LIN {X 0,Y 358.327,Z 844.562,A -85,B 0,C 180,E1 17293.72,E2 17293.72} C_VEL
LIN {X 0,Y 357.15,Z 856.767,A -85,B 0,C 180,E1 17291.793,E2 17291.793} C_VEL
LIN {X 0,Y 356.13,Z 867.565,A -85,B 0,C 180,E1 17289.698,E2 17289.698} C_VEL
LIN {X 0,Y 355.243,Z 877.441,A -85,B 0,C 180,E1 17287.277,E2 17287.277} C_VEL
LIN {X 0,Y 354.65,Z 885.167,A -85,B 0,C 180,E1 17284.852,E2 17284.852} C_VEL
LIN {X 0,Y 354.297,Z 891.351,A -85,B 0,C 180,E1 17282.265,E2 17282.265} C_VEL
LIN {X 0,Y 354.201,Z 895.635,A -85,B 0,C 180,E1 17279.677,E2 17279.677} C_VEL
LIN {X 0,Y 354.349,Z 898.233,A -85,B 0,C 180,E1 17277.089,E2 17277.089} C_VEL
LIN {X 0,Y 354.713,Z 899.091,A -85,B 0,C 180,E1 17274.501,E2 17274.501} C_VEL
LIN {X 0,Y 355.419,Z 898.216,A -85,B 0,C 180,E1 17271.751,E2 17271.751} C_VEL
LIN {X 0,Y 356.484,Z 895.398,A -85,B 0,C 180,E1 17269.005,E2 17269.005} C_VEL
LIN {X 0,Y 357.89,Z 890.872,A -85,B 0,C 180,E1 17266.428,E2 17266.428} C_VEL
LIN {X 0,Y 359.589,Z 884.914,A -85,B 0,C 180,E1 17264.022,E2 17264.022} C_VEL
LIN {X 0,Y 361.837,Z 876.313,A -85,B 0,C 180,E1 17261.472,E2 17261.472} C_VEL
LIN {X 0,Y 364.2,Z 866.559,A -85,B 0,C 180,E1 17259.259,E2 17259.259} C_VEL
LIN {X 0,Y 366.508,Z 856.117,A -85,B 0,C 180,E1 17257.378,E2 17257.378} C_VEL
LIN {X 0,Y 368.84,Z 844.36,A -85,B 0,C 180,E1 17255.667,E2 17255.667} C_VEL
LIN {X 0,Y 371.242,Z 830.372,A -85,B 0,C 180,E1 17254.046,E2 17254.046} C_VEL
LIN {X 0,Y 373.396,Z 815.063,A -85,B 0,C 180,E1 17252.663,E2 17252.663} C_VEL
LIN {X 0,Y 375.26,Z 798.255,A -85,B 0,C 180,E1 17251.515,E2 17251.515} C_VEL
LIN {X 0,Y 379.041,Z 772.114,A -85,B 0,C 180,E1 17250.009,E2 17250.009} C_VEL
LIN {X 0,Y 387.538,Z 729.748,A -85,B 0,C 180,E1 17247.894,E2 17247.894} C_VEL
LIN {X 0,Y 397.033,Z 682.025,A -85,B 0,C 180,E1 17245.846,E2 17245.846} C_VEL
LIN {X 0,Y 397.784,Z 679.73,A -85,B 0,C 180,E1 17245.734,E2 17245.734} C_VEL
LIN {X 0,Y 407.089,Z 665.776,A -85,B 0,C 180,E1 17244.661,E2 17244.661} C_VEL
LIN {X 0,Y 408.416,Z 663.697,A -85,B 0,C 180,E1 17244.363,E2 17244.363} C_VEL
LIN {X 0,Y 415.736,Z 652.988,A -85,B 0,C 180,E1 17242.392,E2 17242.392} C_VEL
LIN {X 0,Y 409.908,Z 662.726,A -85,B 0,C 180,E1 17240.427,E2 17240.427} C_VEL
LIN {X 0,Y 406.103,Z 673.236,A -85,B 0,C 180,E1 17238.247,E2 17238.247} C_VEL
LIN {X 0,Y 404.763,Z 684.168,A -85,B 0,C 180,E1 17235.96,E2 17235.96} C_VEL
LIN {X 0,Y 406.043,Z 694.968,A -85,B 0,C 180,E1 17233.72,E2 17233.72} C_VEL
LIN {X 0,Y 408.323,Z 702.84,A -85,B 0,C 180,E1 17232.141,E2 17232.141} C_VEL
LIN {X 0,Y 398.65,Z 721.921,A -85,B 0,C 180,E1 17231.177,E2 17231.177} C_VEL
LIN {X 0,Y 396.234,Z 727.339,A -85,B 0,C 180,E1 17230.919,E2 17230.919} C_VEL
LIN {X 0,Y 391.082,Z 751.783,A -85,B 0,C 180,E1 17230.609,E2 17230.609} C_VEL
LIN {X 0,Y 389.402,Z 762.099,A -85,B 0,C 180,E1 17230.457,E2 17230.457} C_VEL
LIN {X 0,Y 387.915,Z 782.543,A -85,B 0,C 180,E1 17230.159,E2 17230.159} C_VEL
LIN {X 0,Y 386.621,Z 805.179,A -85,B 0,C 180,E1 17229.634,E2 17229.634} C_VEL
LIN {X 0,Y 384.476,Z 826.222,A -85,B 0,C 180,E1 17228.907,E2 17228.907} C_VEL
LIN {X 0,Y 381.713,Z 846.978,A -85,B 0,C 180,E1 17227.898,E2 17227.898} C_VEL
LIN {X 0,Y 378.758,Z 865.544,A -85,B 0,C 180,E1 17226.722,E2 17226.722} C_VEL
LIN {X 0,Y 375.32,Z 884.39,A -85,B 0,C 180,E1 17225.224,E2 17225.224} C_VEL
LIN {X 0,Y 371.531,Z 902.981,A -85,B 0,C 180,E1 17223.392,E2 17223.392} C_VEL
LIN {X 0,Y 367.741,Z 920.372,A -85,B 0,C 180,E1 17221.287,E2 17221.287} C_VEL
LIN {X 0,Y 364.185,Z 936.094,A -85,B 0,C 180,E1 17218.986,E2 17218.986} C_VEL
LIN {X 0,Y 360.968,Z 950.344,A -85,B 0,C 180,E1 17216.486,E2 17216.486} C_VEL
LIN {X 0,Y 358.088,Z 963.562,A -85,B 0,C 180,E1 17213.709,E2 17213.709} C_VEL
LIN {X 0,Y 355.694,Z 975.773,A -85,B 0,C 180,E1 17210.6,E2 17210.6} C_VEL
LIN {X 0,Y 353.976,Z 985.945,A -85,B 0,C 180,E1 17207.423,E2 17207.423} C_VEL
LIN {X 0,Y 352.891,Z 994.085,A -85,B 0,C 180,E1 17204.271,E2 17204.271} C_VEL
LIN {X 0,Y 352.346,Z 1000.464,A -85,B 0,C 180,E1 17201.127,E2 17201.127} C_VEL
LIN {X 0,Y 352.156,Z 1005.337,A -85,B 0,C 180,E1 17197.834,E2 17197.834} C_VEL
LIN {X 0,Y 352.163,Z 1008.374,A -85,B 0,C 180,E1 17194.724,E2 17194.724} C_VEL
LIN {X 0,Y 352.223,Z 1009.946,A -85,B 0,C 180,E1 17191.628,E2 17191.628} C_VEL
LIN {X 0,Y 352.225,Z 1009.994,A -85,B 0,C 180,E1 17188.7,E2 17188.7} C_VEL
LIN {X 0,Y 352.165,Z 1008.606,A -85,B 0,C 180,E1 17185.604,E2 17185.604} C_VEL
LIN {X 0,Y 352.117,Z 1005.756,A -85,B 0,C 180,E1 17182.495,E2 17182.495} C_VEL
LIN {X 0,Y 352.294,Z 1001.017,A -85,B 0,C 180,E1 17179.205,E2 17179.205} C_VEL
LIN {X 0,Y 352.795,Z 994.807,A -85,B 0,C 180,E1 17176.061,E2 17176.061} C_VEL
LIN {X 0,Y 353.805,Z 986.872,A -85,B 0,C 180,E1 17172.909,E2 17172.909} C_VEL
LIN {X 0,Y 355.418,Z 977.017,A -85,B 0,C 180,E1 17169.757,E2 17169.757} C_VEL
LIN {X 0,Y 357.478,Z 966.389,A -85,B 0,C 180,E1 17166.948,E2 17166.948} C_VEL
LIN {X 0,Y 360.351,Z 953.009,A -85,B 0,C 180,E1 17164.026,E2 17164.026} C_VEL
LIN {X 0,Y 363.681,Z 938.075,A -85,B 0,C 180,E1 17161.332,E2 17161.332} C_VEL
LIN {X 0,Y 367.303,Z 922.064,A -85,B 0,C 180,E1 17158.947,E2 17158.947} C_VEL
LIN {X 0,Y 370.863,Z 905.617,A -85,B 0,C 180,E1 17156.912,E2 17156.912} C_VEL
LIN {X 0,Y 374.426,Z 888.379,A -85,B 0,C 180,E1 17155.149,E2 17155.149} C_VEL
LIN {X 0,Y 377.967,Z 869.449,A -85,B 0,C 180,E1 17153.568,E2 17153.568} C_VEL
LIN {X 0,Y 381.074,Z 850.673,A -85,B 0,C 180,E1 17152.314,E2 17152.314} C_VEL
LIN {X 0,Y 383.853,Z 830.914,A -85,B 0,C 180,E1 17151.292,E2 17151.292} C_VEL
LIN {X 0,Y 386.143,Z 809.808,A -85,B 0,C 180,E1 17150.496,E2 17150.496} C_VEL
LIN {X 0,Y 387.604,Z 787.894,A -85,B 0,C 180,E1 17149.946,E2 17149.946} C_VEL
LIN {X 0,Y 388.886,Z 765.567,A -85,B 0,C 180,E1 17149.574,E2 17149.574} C_VEL
LIN {X 0,Y 392.068,Z 738.697,A -85,B 0,C 180,E1 17149.337,E2 17149.337} C_VEL
LIN {X 0,Y 394.002,Z 728.374,A -85,B 0,C 180,E1 17149.294,E2 17149.294} C_VEL
LIN {X 0,Y 406.256,Z 703.937,A -85,B 0,C 180,E1 17147.978,E2 17147.978} C_VEL
LIN {X 0,Y 407.296,Z 701.642,A -85,B 0,C 180,E1 17147.848,E2 17147.848} C_VEL
LIN {X 0,Y 400.592,Z 686.213,A -85,B 0,C 180,E1 17145.753,E2 17145.753} C_VEL
LIN {X 0,Y 395.618,Z 668.635,A -85,B 0,C 180,E1 17143.504,E2 17143.504} C_VEL
LIN {X 0,Y 392.777,Z 649.847,A -85,B 0,C 180,E1 17141.247,E2 17141.247} C_VEL
LIN {X 0,Y 392.112,Z 630.144,A -85,B 0,C 180,E1 17139.038,E2 17139.038} C_VEL
LIN {X 0,Y 393.724,Z 606.831,A -85,B 0,C 180,E1 17136.634,E2 17136.634} C_VEL
LIN {X 0,Y 400.166,Z 566.042,A -85,B 0,C 180,E1 17132.748,E2 17132.748} C_VEL
LIN {X 0,Y 391.222,Z 546.366,A -85,B 0,C 180,E1 17129.051,E2 17129.051} C_VEL
LIN {X 0,Y 382.764,Z 528.585,A -85,B 0,C 180,E1 17125.366,E2 17125.366} C_VEL
LIN {X 0,Y 374.331,Z 511.509,A -85,B 0,C 180,E1 17121.465,E2 17121.465} C_VEL
LIN {X 0,Y 367.669,Z 498.547,A -85,B 0,C 180,E1 17118.224,E2 17118.224} C_VEL
LIN {X 0,Y 362.734,Z 489.046,A -85,B 0,C 180,E1 17115.672,E2 17115.672} C_VEL
LIN {X 0,Y 360.463,Z 484.681,A -85,B 0,C 180,E1 17114.456,E2 17114.456} C_VEL
LIN {X 0,Y 357.931,Z 479.938,A -85,B 0,C 180,E1 17113.077,E2 17113.077} C_VEL
LIN {X 0,Y 355.754,Z 475.696,A -85,B 0,C 180,E1 17111.839,E2 17111.839} C_VEL
LIN {X 0,Y 354.097,Z 472.685,A -85,B 0,C 180,E1 17110.905,E2 17110.905} C_VEL
LIN {X 0,Y 353.827,Z 471.413,A -85,B 0,C 180,E1 17110.584,E2 17110.584} C_VEL
LIN {X 0,Y 353.868,Z 471.408,A -85,B 0,C 180,E1 17106.489,E2 17106.489} C_VEL
LIN {X 0,Y 353.825,Z 471.412,A -85,B 0,C 180,E1 17102.267,E2 17102.267} C_VEL
LIN {X 0,Y 353.866,Z 471.403,A -85,B 0,C 180,E1 17098.219,E2 17098.219} C_VEL
LIN {X 0,Y 353.825,Z 471.407,A -85,B 0,C 180,E1 17093.998,E2 17093.998} C_VEL
LIN {X 0,Y 353.864,Z 471.405,A -85,B 0,C 180,E1 17089.91,E2 17089.91} C_VEL
LIN {X 0,Y 353.822,Z 471.397,A -85,B 0,C 180,E1 17085.6,E2 17085.6} C_VEL
LIN {X 0,Y 353.864,Z 471.384,A -85,B 0,C 180,E1 17081.551,E2 17081.551} C_VEL
LIN {X 0,Y 353.822,Z 471.39,A -85,B 0,C 180,E1 17077.398,E2 17077.398} C_VEL
LIN {X 0,Y 353.865,Z 471.389,A -85,B 0,C 180,E1 17073.234,E2 17073.234} C_VEL
LIN {X 0,Y 353.823,Z 471.397,A -85,B 0,C 180,E1 17069.048,E2 17069.048} C_VEL
LIN {X 0,Y 353.862,Z 471.507,A -85,B 0,C 180,E1 17067.193,E2 17067.193} C_VEL
LIN {X 0,Y 355.032,Z 474.666,A -85,B 0,C 180,E1 17066.47,E2 17066.47} C_VEL
LIN {X 0,Y 356.9,Z 476.875,A -85,B 0,C 180,E1 17065.729,E2 17065.729} C_VEL
LIN {X 0,Y 358.818,Z 480.752,A -85,B 0,C 180,E1 17064.773,E2 17064.773} C_VEL
LIN {X 0,Y 359.911,Z 482.426,A -85,B 0,C 180,E1 17064.31,E2 17064.31} C_VEL
LIN {X 0,Y 365.518,Z 492.86,A -85,B 0,C 180,E1 17061.814,E2 17061.814} C_VEL
LIN {X 0,Y 371.605,Z 504.363,A -85,B 0,C 180,E1 17059.328,E2 17059.328} C_VEL
LIN {X 0,Y 382.76,Z 521.472,A -85,B 0,C 180,E1 17056.939,E2 17056.939} C_VEL
LIN {X 0,Y 393.149,Z 539.114,A -85,B 0,C 180,E1 17054.878,E2 17054.878} C_VEL
LIN {X 0,Y 397.29,Z 547.107,A -85,B 0,C 180,E1 17054.083,E2 17054.083} C_VEL
LIN {X 0,Y 388.766,Z 764.74,A -85,B 0,C 180,E1 17049.883,E2 17049.883} C_VEL
LIN {X 0,Y 387.23,Z 785.322,A -85,B 0,C 180,E1 17049.247,E2 17049.247} C_VEL
LIN {X 0,Y 385.016,Z 805.804,A -85,B 0,C 180,E1 17048.346,E2 17048.346} C_VEL
LIN {X 0,Y 382.432,Z 824.71,A -85,B 0,C 180,E1 17047.246,E2 17047.246} C_VEL
LIN {X 0,Y 379.409,Z 843.123,A -85,B 0,C 180,E1 17045.898,E2 17045.898} C_VEL
LIN {X 0,Y 375.891,Z 861.453,A -85,B 0,C 180,E1 17044.234,E2 17044.234} C_VEL
LIN {X 0,Y 372.225,Z 878.68,A -85,B 0,C 180,E1 17042.312,E2 17042.312} C_VEL
LIN {X 0,Y 368.616,Z 894.311,A -85,B 0,C 180,E1 17040.208,E2 17040.208} C_VEL
LIN {X 0,Y 365.189,Z 908.557,A -85,B 0,C 180,E1 17037.916,E2 17037.916} C_VEL
LIN {X 0,Y 361.934,Z 921.884,A -85,B 0,C 180,E1 17035.352,E2 17035.352} C_VEL
LIN {X 0,Y 359.073,Z 933.808,A -85,B 0,C 180,E1 17032.597,E2 17032.597} C_VEL
LIN {X 0,Y 356.646,Z 944.461,A -85,B 0,C 180,E1 17029.613,E2 17029.613} C_VEL
LIN {X 0,Y 354.714,Z 953.775,A -85,B 0,C 180,E1 17026.371,E2 17026.371} C_VEL
LIN {X 0,Y 353.405,Z 961.197,A -85,B 0,C 180,E1 17023.081,E2 17023.081} C_VEL
LIN {X 0,Y 352.629,Z 966.798,A -85,B 0,C 180,E1 17019.794,E2 17019.794} C_VEL
LIN {X 0,Y 352.248,Z 970.723,A -85,B 0,C 180,E1 17016.519,E2 17016.519} C_VEL
LIN {X 0,Y 352.161,Z 971.831,A -85,B 0,C 180,E1 17015.277,E2 17015.277} C_VEL
LIN {X 0,Y 351.121,Z 972.736,A -85,B 0,C 180,E1 17014.032,E2 17014.032} C_VEL
LIN {X 0,Y 346.458,Z 973.982,A -85,B 0,C 180,E1 17011.675,E2 17011.675} C_VEL
LIN {X 0,Y 344.214,Z 974.308,A -85,B 0,C 180,E1 17010.044,E2 17010.044} C_VEL
LIN {X 0,Y 344.066,Z 974.269,A -85,B 0,C 180,E1 17009.579,E2 17009.579} C_VEL
LIN {X 0,Y 344.109,Z 973.398,A -85,B 0,C 180,E1 17006.334,E2 17006.334} C_VEL
LIN {X 0,Y 344.298,Z 970.92,A -85,B 0,C 180,E1 17002.993,E2 17002.993} C_VEL
LIN {X 0,Y 344.737,Z 966.862,A -85,B 0,C 180,E1 16999.64,E2 16999.64} C_VEL
LIN {X 0,Y 345.615,Z 961.121,A -85,B 0,C 180,E1 16996.276,E2 16996.276} C_VEL
LIN {X 0,Y 346.993,Z 953.972,A -85,B 0,C 180,E1 16993.07,E2 16993.07} C_VEL
LIN {X 0,Y 348.982,Z 945.03,A -85,B 0,C 180,E1 16989.89,E2 16989.89} C_VEL
LIN {X 0,Y 351.675,Z 933.95,A -85,B 0,C 180,E1 16986.721,E2 16986.721} C_VEL
LIN {X 0,Y 354.725,Z 921.962,A -85,B 0,C 180,E1 16983.913,E2 16983.913} C_VEL
LIN {X 0,Y 358.171,Z 908.563,A -85,B 0,C 180,E1 16981.304,E2 16981.304} C_VEL
LIN {X 0,Y 361.933,Z 893.686,A -85,B 0,C 180,E1 16978.895,E2 16978.895} C_VEL
LIN {X 0,Y 365.672,Z 878.113,A -85,B 0,C 180,E1 16976.793,E2 16976.793} C_VEL
LIN {X 0,Y 369.445,Z 861.121,A -85,B 0,C 180,E1 16974.892,E2 16974.892} C_VEL
LIN {X 0,Y 373.11,Z 842.762,A -85,B 0,C 180,E1 16973.215,E2 16973.215} C_VEL
LIN {X 0,Y 376.295,Z 824.075,A -85,B 0,C 180,E1 16971.845,E2 16971.845} C_VEL
LIN {X 0,Y 379.033,Z 804.56,A -85,B 0,C 180,E1 16970.72,E2 16970.72} C_VEL
LIN {X 0,Y 381.218,Z 784.635,A -85,B 0,C 180,E1 16969.854,E2 16969.854} C_VEL
LIN {X 0,Y 382.807,Z 763.298,A -85,B 0,C 180,E1 16969.208,E2 16969.208} C_VEL
LIN {X 0,Y 391.184,Z 555.703,A -85,B 0,C 180,E1 16965.148,E2 16965.148} C_VEL
LIN {X 0,Y 382.835,Z 539.982,A -85,B 0,C 180,E1 16963.461,E2 16963.461} C_VEL
LIN {X 0,Y 372.499,Z 522.649,A -85,B 0,C 180,E1 16961.247,E2 16961.247} C_VEL
LIN {X 0,Y 368.988,Z 517.5,A -85,B 0,C 180,E1 16960.465,E2 16960.465} C_VEL
LIN {X 0,Y 366.654,Z 518.374,A -85,B 0,C 180,E1 16960.059,E2 16960.059} C_VEL
LIN {X 0,Y 364.475,Z 517.811,A -85,B 0,C 180,E1 16959.629,E2 16959.629} C_VEL
LIN {X 0,Y 364.222,Z 517.629,A -85,B 0,C 180,E1 16959.56,E2 16959.56} C_VEL
LIN {X 0,Y 370.358,Z 535.71,A -85,B 0,C 180,E1 16956.174,E2 16956.174} C_VEL
LIN {X 0,Y 371.873,Z 541.268,A -85,B 0,C 180,E1 16955.221,E2 16955.221} C_VEL
LIN {X 0,Y 367.71,Z 575.018,A -85,B 0,C 180,E1 16951.107,E2 16951.107} C_VEL
LIN {X 0,Y 363.77,Z 611.009,A -85,B 0,C 180,E1 16946.793,E2 16946.793} C_VEL
LIN {X 0,Y 361.959,Z 630.785,A -85,B 0,C 180,E1 16944.502,E2 16944.502} C_VEL
LIN {X 0,Y 362.358,Z 637.138,A -85,B 0,C 180,E1 16944.255,E2 16944.255} C_VEL
LIN {X 0,Y 355.628,Z 765.283,A -85,B 0,C 180,E1 16940.307,E2 16940.307} C_VEL
LIN {X 0,Y 355.062,Z 783.346,A -85,B 0,C 180,E1 16939.585,E2 16939.585} C_VEL
LIN {X 0,Y 354.204,Z 800.194,A -85,B 0,C 180,E1 16938.602,E2 16938.602} C_VEL
LIN {X 0,Y 353.149,Z 815.686,A -85,B 0,C 180,E1 16937.38,E2 16937.38} C_VEL
LIN {X 0,Y 351.952,Z 830.328,A -85,B 0,C 180,E1 16935.911,E2 16935.911} C_VEL
LIN {X 0,Y 350.574,Z 845.108,A -85,B 0,C 180,E1 16934.03,E2 16934.03} C_VEL
LIN {X 0,Y 349.35,Z 857.47,A -85,B 0,C 180,E1 16932.06,E2 16932.06} C_VEL
LIN {X 0,Y 348.283,Z 868.348,A -85,B 0,C 180,E1 16929.919,E2 16929.919} C_VEL
LIN {X 0,Y 347.408,Z 877.732,A -85,B 0,C 180,E1 16927.608,E2 16927.608} C_VEL
LIN {X 0,Y 346.779,Z 885.724,A -85,B 0,C 180,E1 16925.128,E2 16925.128} C_VEL
LIN {X 0,Y 346.389,Z 892.109,A -85,B 0,C 180,E1 16922.482,E2 16922.482} C_VEL
LIN {X 0,Y 346.293,Z 896.653,A -85,B 0,C 180,E1 16919.835,E2 16919.835} C_VEL
LIN {X 0,Y 346.458,Z 899.551,A -85,B 0,C 180,E1 16917.023,E2 16917.023} C_VEL
LIN {X 0,Y 346.867,Z 900.541,A -85,B 0,C 180,E1 16914.376,E2 16914.376} C_VEL
LIN {X 0,Y 347.635,Z 899.778,A -85,B 0,C 180,E1 16911.565,E2 16911.565} C_VEL
LIN {X 0,Y 348.881,Z 896.874,A -85,B 0,C 180,E1 16908.595,E2 16908.595} C_VEL
LIN {X 0,Y 350.434,Z 892.375,A -85,B 0,C 180,E1 16905.955,E2 16905.955} C_VEL
LIN {X 0,Y 352.411,Z 885.971,A -85,B 0,C 180,E1 16903.348,E2 16903.348} C_VEL
LIN {X 0,Y 354.739,Z 877.962,A -85,B 0,C 180,E1 16900.916,E2 16900.916} C_VEL
LIN {X 0,Y 357.498,Z 867.558,A -85,B 0,C 180,E1 16898.508,E2 16898.508} C_VEL
LIN {X 0,Y 360.338,Z 855.603,A -85,B 0,C 180,E1 16896.362,E2 16896.362} C_VEL
LIN {X 0,Y 363.15,Z 842.283,A -85,B 0,C 180,E1 16894.476,E2 16894.476} C_VEL
LIN {X 0,Y 365.813,Z 827.572,A -85,B 0,C 180,E1 16892.842,E2 16892.842} C_VEL
LIN {X 0,Y 368.218,Z 811.346,A -85,B 0,C 180,E1 16891.451,E2 16891.451} C_VEL
LIN {X 0,Y 371.798,Z 786.102,A -85,B 0,C 180,E1 16889.809,E2 16889.809} C_VEL
LIN {X 0,Y 378.125,Z 755.401,A -85,B 0,C 180,E1 16888.072,E2 16888.072} C_VEL
LIN {X 0,Y 388.531,Z 709.223,A -85,B 0,C 180,E1 16885.875,E2 16885.875} C_VEL
LIN {X 0,Y 394.034,Z 683.55,A -85,B 0,C 180,E1 16884.794,E2 16884.794} C_VEL
LIN {X 0,Y 403.144,Z 670.374,A -85,B 0,C 180,E1 16883.824,E2 16883.824} C_VEL
LIN {X 0,Y 404.573,Z 668.344,A -85,B 0,C 180,E1 16883.621,E2 16883.621} C_VEL
LIN {X 0,Y 409.42,Z 661.58,A -85,B 0,C 180,E1 16882.355,E2 16882.355} C_VEL
LIN {X 0,Y 403.832,Z 671.327,A -85,B 0,C 180,E1 16880.299,E2 16880.299} C_VEL
LIN {X 0,Y 400.331,Z 682.047,A -85,B 0,C 180,E1 16877.983,E2 16877.983} C_VEL
LIN {X 0,Y 399.464,Z 692.505,A -85,B 0,C 180,E1 16875.707,E2 16875.707} C_VEL
LIN {X 0,Y 401.087,Z 702.877,A -85,B 0,C 180,E1 16873.476,E2 16873.476} C_VEL
LIN {X 0,Y 401.753,Z 705.735,A -85,B 0,C 180,E1 16872.897,E2 16872.897} C_VEL
LIN {X 0,Y 392.641,Z 724.079,A -85,B 0,C 180,E1 16871.958,E2 16871.958} C_VEL
LIN {X 0,Y 386.129,Z 754.105,A -85,B 0,C 180,E1 16871.548,E2 16871.548} C_VEL
LIN {X 0,Y 382.336,Z 772.967,A -85,B 0,C 180,E1 16871.095,E2 16871.095} C_VEL
LIN {X 0,Y 380.859,Z 800.177,A -85,B 0,C 180,E1 16870.537,E2 16870.537} C_VEL
LIN {X 0,Y 378.856,Z 821.051,A -85,B 0,C 180,E1 16869.871,E2 16869.871} C_VEL
LIN {X 0,Y 376.169,Z 841.391,A -85,B 0,C 180,E1 16868.949,E2 16868.949} C_VEL
LIN {X 0,Y 373.036,Z 860.888,A -85,B 0,C 180,E1 16867.768,E2 16867.768} C_VEL
LIN {X 0,Y 369.564,Z 879.545,A -85,B 0,C 180,E1 16866.336,E2 16866.336} C_VEL
LIN {X 0,Y 365.687,Z 898.153,A -85,B 0,C 180,E1 16864.566,E2 16864.566} C_VEL
LIN {X 0,Y 361.789,Z 915.443,A -85,B 0,C 180,E1 16862.551,E2 16862.551} C_VEL
LIN {X 0,Y 358.126,Z 931.067,A -85,B 0,C 180,E1 16860.355,E2 16860.355} C_VEL
LIN {X 0,Y 354.644,Z 945.642,A -85,B 0,C 180,E1 16857.906,E2 16857.906} C_VEL
LIN {X 0,Y 351.397,Z 959.56,A -85,B 0,C 180,E1 16855.086,E2 16855.086} C_VEL
LIN {X 0,Y 348.707,Z 971.862,A -85,B 0,C 180,E1 16852.064,E2 16852.064} C_VEL
LIN {X 0,Y 346.719,Z 982.059,A -85,B 0,C 180,E1 16849.019,E2 16849.019} C_VEL
LIN {X 0,Y 345.336,Z 990.862,A -85,B 0,C 180,E1 16845.794,E2 16845.794} C_VEL
LIN {X 0,Y 344.516,Z 998.173,A -85,B 0,C 180,E1 16842.403,E2 16842.403} C_VEL
LIN {X 0,Y 344.187,Z 1003.425,A -85,B 0,C 180,E1 16839.195,E2 16839.195} C_VEL
LIN {X 0,Y 344.149,Z 1007.041,A -85,B 0,C 180,E1 16836.004,E2 16836.004} C_VEL
LIN {X 0,Y 344.208,Z 1009.106,A -85,B 0,C 180,E1 16832.831,E2 16832.831} C_VEL
LIN {X 0,Y 344.244,Z 1009.723,A -85,B 0,C 180,E1 16829.668,E2 16829.668} C_VEL
LIN {X 0,Y 344.196,Z 1008.891,A -85,B 0,C 180,E1 16826.67,E2 16826.67} C_VEL
LIN {X 0,Y 344.145,Z 1006.54,A -85,B 0,C 180,E1 16823.495,E2 16823.495} C_VEL
LIN {X 0,Y 344.219,Z 1002.436,A -85,B 0,C 180,E1 16820.133,E2 16820.133} C_VEL
LIN {X 0,Y 344.605,Z 996.915,A -85,B 0,C 180,E1 16816.921,E2 16816.921} C_VEL
LIN {X 0,Y 345.55,Z 989.188,A -85,B 0,C 180,E1 16813.528,E2 16813.528} C_VEL
LIN {X 0,Y 347.065,Z 979.934,A -85,B 0,C 180,E1 16810.303,E2 16810.303} C_VEL
LIN {X 0,Y 349.235,Z 969.022,A -85,B 0,C 180,E1 16807.202,E2 16807.202} C_VEL
LIN {X 0,Y 352.042,Z 956.398,A -85,B 0,C 180,E1 16804.245,E2 16804.245} C_VEL
LIN {X 0,Y 355.234,Z 942.818,A -85,B 0,C 180,E1 16801.598,E2 16801.598} C_VEL
LIN {X 0,Y 358.829,Z 927.815,A -85,B 0,C 180,E1 16799.157,E2 16799.157} C_VEL
LIN {X 0,Y 362.69,Z 911.261,A -85,B 0,C 180,E1 16796.919,E2 16796.919} C_VEL
LIN {X 0,Y 366.607,Z 893.632,A -85,B 0,C 180,E1 16794.964,E2 16794.964} C_VEL
LIN {X 0,Y 370.389,Z 874.916,A -85,B 0,C 180,E1 16793.279,E2 16793.279} C_VEL
LIN {X 0,Y 373.723,Z 856.216,A -85,B 0,C 180,E1 16791.927,E2 16791.927} C_VEL
LIN {X 0,Y 376.714,Z 836.78,A -85,B 0,C 180,E1 16790.826,E2 16790.826} C_VEL
LIN {X 0,Y 379.295,Z 816.001,A -85,B 0,C 180,E1 16789.951,E2 16789.951} C_VEL
LIN {X 0,Y 381.074,Z 795.371,A -85,B 0,C 180,E1 16789.345,E2 16789.345} C_VEL
LIN {X 0,Y 382.505,Z 769.105,A -85,B 0,C 180,E1 16788.848,E2 16788.848} C_VEL
LIN {X 0,Y 385.797,Z 739.934,A -85,B 0,C 180,E1 16788.569,E2 16788.569} C_VEL
LIN {X 0,Y 388.428,Z 725.254,A -85,B 0,C 180,E1 16788.534,E2 16788.534} C_VEL
LIN {X 0,Y 399.359,Z 703.372,A -85,B 0,C 180,E1 16787.325,E2 16787.325} C_VEL
LIN {X 0,Y 392.97,Z 687.667,A -85,B 0,C 180,E1 16785.189,E2 16785.189} C_VEL
LIN {X 0,Y 388.217,Z 669.39,A -85,B 0,C 180,E1 16782.838,E2 16782.838} C_VEL
LIN {X 0,Y 385.707,Z 649.996,A -85,B 0,C 180,E1 16780.493,E2 16780.493} C_VEL
LIN {X 0,Y 385.416,Z 629.38,A -85,B 0,C 180,E1 16778.183,E2 16778.183} C_VEL
LIN {X 0,Y 387.601,Z 604.874,A -85,B 0,C 180,E1 16775.653,E2 16775.653} C_VEL
LIN {X 0,Y 393.478,Z 569.598,A -85,B 0,C 180,E1 16772.251,E2 16772.251} C_VEL
LIN {X 0,Y 384.721,Z 550.197,A -85,B 0,C 180,E1 16768.548,E2 16768.548} C_VEL
LIN {X 0,Y 376.279,Z 532.557,A -85,B 0,C 180,E1 16764.824,E2 16764.824} C_VEL
LIN {X 0,Y 368.499,Z 516.647,A -85,B 0,C 180,E1 16761.154,E2 16761.154} C_VEL
LIN {X 0,Y 361.87,Z 503.689,A -85,B 0,C 180,E1 16757.86,E2 16757.86} C_VEL
LIN {X 0,Y 356.908,Z 494.103,A -85,B 0,C 180,E1 16755.268,E2 16755.268} C_VEL
LIN {X 0,Y 352.715,Z 485.947,A -85,B 0,C 180,E1 16752.941,E2 16752.941} C_VEL
LIN {X 0,Y 350.217,Z 481.279,A -85,B 0,C 180,E1 16751.528,E2 16751.528} C_VEL
LIN {X 0,Y 347.771,Z 476.632,A -85,B 0,C 180,E1 16750.1,E2 16750.1} C_VEL
LIN {X 0,Y 346.169,Z 473.606,A -85,B 0,C 180,E1 16749.14,E2 16749.14} C_VEL
LIN {X 0,Y 345.916,Z 472.397,A -85,B 0,C 180,E1 16748.812,E2 16748.812} C_VEL
LIN {X 0,Y 345.91,Z 472.397,A -85,B 0,C 180,E1 16744.642,E2 16744.642} C_VEL
LIN {X 0,Y 345.917,Z 472.394,A -85,B 0,C 180,E1 16740.165,E2 16740.165} C_VEL
LIN {X 0,Y 345.892,Z 472.395,A -85,B 0,C 180,E1 16736.022,E2 16736.022} C_VEL
LIN {X 0,Y 345.917,Z 472.369,A -85,B 0,C 180,E1 16731.69,E2 16731.69} C_VEL
LIN {X 0,Y 345.891,Z 472.377,A -85,B 0,C 180,E1 16727.648,E2 16727.648} C_VEL
LIN {X 0,Y 345.919,Z 472.385,A -85,B 0,C 180,E1 16723.372,E2 16723.372} C_VEL
LIN {X 0,Y 345.891,Z 472.4,A -85,B 0,C 180,E1 16719.172,E2 16719.172} C_VEL
LIN {X 0,Y 345.926,Z 472.397,A -85,B 0,C 180,E1 16714.856,E2 16714.856} C_VEL
LIN {X 0,Y 345.897,Z 472.4,A -85,B 0,C 180,E1 16710.567,E2 16710.567} C_VEL
LIN {X 0,Y 345.888,Z 472.397,A -85,B 0,C 180,E1 16709.151,E2 16709.151} C_VEL
LIN {X 0,Y 347.044,Z 475.6,A -85,B 0,C 180,E1 16708.375,E2 16708.375} C_VEL
LIN {X 0,Y 349.2,Z 478.304,A -85,B 0,C 180,E1 16707.432,E2 16707.432} C_VEL
LIN {X 0,Y 351.081,Z 481.889,A -85,B 0,C 180,E1 16706.461,E2 16706.461} C_VEL
LIN {X 0,Y 352.18,Z 483.366,A -85,B 0,C 180,E1 16705.993,E2 16705.993} C_VEL
LIN {X 0,Y 357.956,Z 493.917,A -85,B 0,C 180,E1 16703.288,E2 16703.288} C_VEL
LIN {X 0,Y 364.46,Z 505.727,A -85,B 0,C 180,E1 16700.623,E2 16700.623} C_VEL
LIN {X 0,Y 375.385,Z 522.241,A -85,B 0,C 180,E1 16698.147,E2 16698.147} C_VEL
LIN {X 0,Y 386.228,Z 540.302,A -85,B 0,C 180,E1 16695.888,E2 16695.888} C_VEL
LIN {X 0,Y 391.461,Z 550.328,A -85,B 0,C 180,E1 16694.84,E2 16694.84} C_VEL
LIN {X 0,Y 382.655,Z 765.265,A -85,B 0,C 180,E1 16690.646,E2 16690.646} C_VEL
LIN {X 0,Y 381.071,Z 785.681,A -85,B 0,C 180,E1 16690.008,E2 16690.008} C_VEL
LIN {X 0,Y 378.76,Z 806.255,A -85,B 0,C 180,E1 16689.094,E2 16689.094} C_VEL
LIN {X 0,Y 376.08,Z 825.101,A -85,B 0,C 180,E1 16687.985,E2 16687.985} C_VEL
LIN {X 0,Y 372.929,Z 843.521,A -85,B 0,C 180,E1 16686.622,E2 16686.622} C_VEL
LIN {X 0,Y 369.262,Z 861.856,A -85,B 0,C 180,E1 16684.937,E2 16684.937} C_VEL
LIN {X 0,Y 365.426,Z 879.088,A -85,B 0,C 180,E1 16682.989,E2 16682.989} C_VEL
LIN {X 0,Y 361.663,Z 894.667,A -85,B 0,C 180,E1 16680.861,E2 16680.861} C_VEL
LIN {X 0,Y 358.042,Z 908.971,A -85,B 0,C 180,E1 16678.523,E2 16678.523} C_VEL
LIN {X 0,Y 354.616,Z 922.3,A -85,B 0,C 180,E1 16675.914,E2 16675.914} C_VEL
LIN {X 0,Y 351.588,Z 934.225,A -85,B 0,C 180,E1 16673.106,E2 16673.106} C_VEL
LIN {X 0,Y 348.943,Z 945.143,A -85,B 0,C 180,E1 16669.973,E2 16669.973} C_VEL
LIN {X 0,Y 346.942,Z 954.193,A -85,B 0,C 180,E1 16666.749,E2 16666.749} C_VEL
LIN {X 0,Y 345.533,Z 961.614,A -85,B 0,C 180,E1 16663.384,E2 16663.384} C_VEL
LIN {X 0,Y 344.694,Z 967.213,A -85,B 0,C 180,E1 16660.022,E2 16660.022} C_VEL
LIN {X 0,Y 344.276,Z 971.146,A -85,B 0,C 180,E1 16656.66,E2 16656.66} C_VEL
LIN {X 0,Y 344.1,Z 973.489,A -85,B 0,C 180,E1 16653.331,E2 16653.331} C_VEL
LIN {X 0,Y 344.077,Z 974.311,A -85,B 0,C 180,E1 16649.999,E2 16649.999} C_VEL
LIN {X 0,Y 344.066,Z 974.269,A -85,B 0,C 180,E1 16649.579,E2 16649.579} C_VEL
LIN {X 0,Y 343.065,Z 974.169,A -85,B 0,C 180,E1 16648.295,E2 16648.295} C_VEL
LIN {X 0,Y 338.32,Z 973.465,A -85,B 0,C 180,E1 16645.779,E2 16645.779} C_VEL
LIN {X 0,Y 336.356,Z 972.546,A -85,B 0,C 180,E1 16644.204,E2 16644.204} C_VEL
LIN {X 0,Y 336.253,Z 972.144,A -85,B 0,C 180,E1 16643.732,E2 16643.732} C_VEL
LIN {X 0,Y 336.667,Z 968.499,A -85,B 0,C 180,E1 16640.253,E2 16640.253} C_VEL
LIN {X 0,Y 337.533,Z 962.87,A -85,B 0,C 180,E1 16636.64,E2 16636.64} C_VEL
LIN {X 0,Y 338.961,Z 955.643,A -85,B 0,C 180,E1 16633.196,E2 16633.196} C_VEL
LIN {X 0,Y 340.975,Z 946.94,A -85,B 0,C 180,E1 16629.934,E2 16629.934} C_VEL
LIN {X 0,Y 343.551,Z 936.831,A -85,B 0,C 180,E1 16626.864,E2 16626.864} C_VEL
LIN {X 0,Y 346.832,Z 924.621,A -85,B 0,C 180,E1 16623.827,E2 16623.827} C_VEL
LIN {X 0,Y 350.364,Z 911.677,A -85,B 0,C 180,E1 16621.164,E2 16621.164} C_VEL
LIN {X 0,Y 354.203,Z 897.339,A -85,B 0,C 180,E1 16618.707,E2 16618.707} C_VEL
LIN {X 0,Y 358.256,Z 881.453,A -85,B 0,C 180,E1 16616.453,E2 16616.453} C_VEL
LIN {X 0,Y 362.21,Z 864.507,A -85,B 0,C 180,E1 16614.473,E2 16614.473} C_VEL
LIN {X 0,Y 365.823,Z 847.483,A -85,B 0,C 180,E1 16612.84,E2 16612.84} C_VEL
LIN {X 0,Y 369.269,Z 828.848,A -85,B 0,C 180,E1 16611.381,E2 16611.381} C_VEL
LIN {X 0,Y 372.193,Z 809.912,A -85,B 0,C 180,E1 16610.203,E2 16610.203} C_VEL
LIN {X 0,Y 374.659,Z 789.845,A -85,B 0,C 180,E1 16609.25,E2 16609.25} C_VEL
LIN {X 0,Y 376.494,Z 768.953,A -85,B 0,C 180,E1 16608.545,E2 16608.545} C_VEL
LIN {X 0,Y 378.172,Z 732.317,A -85,B 0,C 180,E1 16607.775,E2 16607.775} C_VEL
LIN {X 0,Y 385.418,Z 558.584,A -85,B 0,C 180,E1 16604.359,E2 16604.359} C_VEL
LIN {X 0,Y 375.654,Z 540.691,A -85,B 0,C 180,E1 16602.304,E2 16602.304} C_VEL
LIN {X 0,Y 367.028,Z 526.362,A -85,B 0,C 180,E1 16600.367,E2 16600.367} C_VEL
LIN {X 0,Y 364.135,Z 526.451,A -85,B 0,C 180,E1 16599.827,E2 16599.827} C_VEL
LIN {X 0,Y 361.345,Z 527.44,A -85,B 0,C 180,E1 16599.321,E2 16599.321} C_VEL
LIN {X 0,Y 359.37,Z 526.749,A -85,B 0,C 180,E1 16598.867,E2 16598.867} C_VEL
LIN {X 0,Y 364.91,Z 543.798,A -85,B 0,C 180,E1 16595.706,E2 16595.706} C_VEL
LIN {X 0,Y 360.636,Z 577.071,A -85,B 0,C 180,E1 16591.601,E2 16591.601} C_VEL
LIN {X 0,Y 356.506,Z 613.339,A -85,B 0,C 180,E1 16587.204,E2 16587.204} C_VEL
LIN {X 0,Y 354.729,Z 631.802,A -85,B 0,C 180,E1 16585.034,E2 16585.034} C_VEL
LIN {X 0,Y 355.1,Z 638.142,A -85,B 0,C 180,E1 16584.784,E2 16584.784} C_VEL
LIN {X 0,Y 348.051,Z 765.418,A -85,B 0,C 180,E1 16580.725,E2 16580.725} C_VEL
LIN {X 0,Y 347.45,Z 784.032,A -85,B 0,C 180,E1 16579.972,E2 16579.972} C_VEL
LIN {X 0,Y 346.532,Z 801.309,A -85,B 0,C 180,E1 16578.942,E2 16578.942} C_VEL
LIN {X 0,Y 345.435,Z 816.73,A -85,B 0,C 180,E1 16577.694,E2 16577.694} C_VEL
LIN {X 0,Y 344.191,Z 831.34,A -85,B 0,C 180,E1 16576.193,E2 16576.193} C_VEL
LIN {X 0,Y 342.82,Z 845.523,A -85,B 0,C 180,E1 16574.354,E2 16574.354} C_VEL
LIN {X 0,Y 341.545,Z 858.048,A -85,B 0,C 180,E1 16572.34,E2 16572.34} C_VEL
LIN {X 0,Y 340.359,Z 869.827,A -85,B 0,C 180,E1 16569.981,E2 16569.981} C_VEL
LIN {X 0,Y 339.471,Z 879.187,A -85,B 0,C 180,E1 16567.617,E2 16567.617} C_VEL
LIN {X 0,Y 338.837,Z 887.172,A -85,B 0,C 180,E1 16565.079,E2 16565.079} C_VEL
LIN {X 0,Y 338.46,Z 893.556,A -85,B 0,C 180,E1 16562.371,E2 16562.371} C_VEL
LIN {X 0,Y 338.379,Z 898.086,A -85,B 0,C 180,E1 16559.662,E2 16559.662} C_VEL
LIN {X 0,Y 338.589,Z 900.999,A -85,B 0,C 180,E1 16556.784,E2 16556.784} C_VEL
LIN {X 0,Y 339.058,Z 901.984,A -85,B 0,C 180,E1 16554.076,E2 16554.076} C_VEL
LIN {X 0,Y 339.918,Z 901.254,A -85,B 0,C 180,E1 16551.202,E2 16551.202} C_VEL
LIN {X 0,Y 341.211,Z 898.6,A -85,B 0,C 180,E1 16548.335,E2 16548.335} C_VEL
LIN {X 0,Y 342.878,Z 894.275,A -85,B 0,C 180,E1 16545.649,E2 16545.649} C_VEL
LIN {X 0,Y 344.982,Z 888.215,A -85,B 0,C 180,E1 16543.029,E2 16543.029} C_VEL
LIN {X 0,Y 347.696,Z 879.691,A -85,B 0,C 180,E1 16540.339,E2 16540.339} C_VEL
LIN {X 0,Y 350.581,Z 869.727,A -85,B 0,C 180,E1 16537.959,E2 16537.959} C_VEL
LIN {X 0,Y 353.634,Z 858.215,A -85,B 0,C 180,E1 16535.797,E2 16535.797} C_VEL
LIN {X 0,Y 356.791,Z 844.747,A -85,B 0,C 180,E1 16533.809,E2 16533.809} C_VEL
LIN {X 0,Y 359.781,Z 829.948,A -85,B 0,C 180,E1 16532.099,E2 16532.099} C_VEL
LIN {X 0,Y 362.312,Z 815.207,A -85,B 0,C 180,E1 16530.761,E2 16530.761} C_VEL
LIN {X 0,Y 366.365,Z 790.602,A -85,B 0,C 180,E1 16529.04,E2 16529.04} C_VEL
LIN {X 0,Y 373.239,Z 760.642,A -85,B 0,C 180,E1 16527.24,E2 16527.24} C_VEL
LIN {X 0,Y 383.716,Z 718.5,A -85,B 0,C 180,E1 16525.148,E2 16525.148} C_VEL
LIN {X 0,Y 390.992,Z 686.986,A -85,B 0,C 180,E1 16523.792,E2 16523.792} C_VEL
LIN {X 0,Y 400.173,Z 674.178,A -85,B 0,C 180,E1 16522.886,E2 16522.886} C_VEL
LIN {X 0,Y 401.394,Z 672.523,A -85,B 0,C 180,E1 16522.75,E2 16522.75} C_VEL
LIN {X 0,Y 403.163,Z 670.175,A -85,B 0,C 180,E1 16522.293,E2 16522.293} C_VEL
LIN {X 0,Y 397.709,Z 680.27,A -85,B 0,C 180,E1 16520.067,E2 16520.067} C_VEL
LIN {X 0,Y 394.674,Z 690.712,A -85,B 0,C 180,E1 16517.711,E2 16517.711} C_VEL
LIN {X 0,Y 394.297,Z 701.06,A -85,B 0,C 180,E1 16515.379,E2 16515.379} C_VEL
LIN {X 0,Y 395.492,Z 708.732,A -85,B 0,C 180,E1 16513.694,E2 16513.694} C_VEL
LIN {X 0,Y 389.401,Z 720.861,A -85,B 0,C 180,E1 16513.08,E2 16513.08} C_VEL
LIN {X 0,Y 387.489,Z 729.939,A -85,B 0,C 180,E1 16512.908,E2 16512.908} C_VEL
LIN {X 0,Y 382.219,Z 753.183,A -85,B 0,C 180,E1 16512.588,E2 16512.588} C_VEL
LIN {X 0,Y 377.964,Z 771.502,A -85,B 0,C 180,E1 16512.115,E2 16512.115} C_VEL
LIN {X 0,Y 375.783,Z 782.234,A -85,B 0,C 180,E1 16511.734,E2 16511.734} C_VEL
LIN {X 0,Y 374.401,Z 804.457,A -85,B 0,C 180,E1 16511.205,E2 16511.205} C_VEL
LIN {X 0,Y 372.086,Z 825.514,A -85,B 0,C 180,E1 16510.464,E2 16510.464} C_VEL
LIN {X 0,Y 369.094,Z 846.229,A -85,B 0,C 180,E1 16509.44,E2 16509.44} C_VEL
LIN {X 0,Y 365.89,Z 864.771,A -85,B 0,C 180,E1 16508.241,E2 16508.241} C_VEL
LIN {X 0,Y 362.142,Z 883.598,A -85,B 0,C 180,E1 16506.71,E2 16506.71} C_VEL
LIN {X 0,Y 358.007,Z 902.178,A -85,B 0,C 180,E1 16504.83,E2 16504.83} C_VEL
LIN {X 0,Y 353.825,Z 919.557,A -85,B 0,C 180,E1 16502.667,E2 16502.667} C_VEL
LIN {X 0,Y 349.896,Z 935.269,A -85,B 0,C 180,E1 16500.29,E2 16500.29} C_VEL
LIN {X 0,Y 346.282,Z 949.511,A -85,B 0,C 180,E1 16497.703,E2 16497.703} C_VEL
LIN {X 0,Y 343.06,Z 962.726,A -85,B 0,C 180,E1 16494.816,E2 16494.816} C_VEL
LIN {X 0,Y 340.424,Z 974.442,A -85,B 0,C 180,E1 16491.721,E2 16491.721} C_VEL
LIN {X 0,Y 338.432,Z 984.462,A -85,B 0,C 180,E1 16488.495,E2 16488.495} C_VEL
LIN {X 0,Y 337.173,Z 992.513,A -85,B 0,C 180,E1 16485.304,E2 16485.304} C_VEL
LIN {X 0,Y 336.434,Z 999.318,A -85,B 0,C 180,E1 16481.834,E2 16481.834} C_VEL
LIN {X 0,Y 336.179,Z 1004.081,A -85,B 0,C 180,E1 16478.553,E2 16478.553} C_VEL
LIN {X 0,Y 336.16,Z 1007.43,A -85,B 0,C 180,E1 16475.12,E2 16475.12} C_VEL
LIN {X 0,Y 336.241,Z 1009.098,A -85,B 0,C 180,E1 16471.875,E2 16471.875} C_VEL
LIN {X 0,Y 336.247,Z 1009.194,A -85,B 0,C 180,E1 16468.808,E2 16468.808} C_VEL
LIN {X 0,Y 336.177,Z 1007.897,A -85,B 0,C 180,E1 16465.566,E2 16465.566} C_VEL
LIN {X 0,Y 336.133,Z 1005.126,A -85,B 0,C 180,E1 16462.308,E2 16462.308} C_VEL
LIN {X 0,Y 336.31,Z 1000.706,A -85,B 0,C 180,E1 16459.032,E2 16459.032} C_VEL
LIN {X 0,Y 336.903,Z 994.329,A -85,B 0,C 180,E1 16455.565,E2 16455.565} C_VEL
LIN {X 0,Y 338.128,Z 986.027,A -85,B 0,C 180,E1 16452.09,E2 16452.09} C_VEL
LIN {X 0,Y 340.018,Z 976.172,A -85,B 0,C 180,E1 16448.797,E2 16448.797} C_VEL
LIN {X 0,Y 342.358,Z 965.544,A -85,B 0,C 180,E1 16445.867,E2 16445.867} C_VEL
LIN {X 0,Y 345.428,Z 952.846,A -85,B 0,C 180,E1 16442.972,E2 16442.972} C_VEL
LIN {X 0,Y 348.962,Z 938.646,A -85,B 0,C 180,E1 16440.286,E2 16440.286} C_VEL
LIN {X 0,Y 352.656,Z 923.932,A -85,B 0,C 180,E1 16437.965,E2 16437.965} C_VEL
LIN {X 0,Y 356.791,Z 906.812,A -85,B 0,C 180,E1 16435.718,E2 16435.718} C_VEL
LIN {X 0,Y 360.82,Z 889.198,A -85,B 0,C 180,E1 16433.827,E2 16433.827} C_VEL
LIN {X 0,Y 364.471,Z 871.672,A -85,B 0,C 180,E1 16432.284,E2 16432.284} C_VEL
LIN {X 0,Y 368.008,Z 852.427,A -85,B 0,C 180,E1 16430.926,E2 16430.926} C_VEL
LIN {X 0,Y 371.049,Z 832.717,A -85,B 0,C 180,E1 16429.858,E2 16429.858} C_VEL
LIN {X 0,Y 373.502,Z 812.539,A -85,B 0,C 180,E1 16429.048,E2 16429.048} C_VEL
LIN {X 0,Y 375.224,Z 791.371,A -85,B 0,C 180,E1 16428.462,E2 16428.462} C_VEL
LIN {X 0,Y 376.627,Z 767.539,A -85,B 0,C 180,E1 16428.03,E2 16428.03} C_VEL
LIN {X 0,Y 379.967,Z 738.755,A -85,B 0,C 180,E1 16427.766,E2 16427.766} C_VEL
LIN {X 0,Y 382.96,Z 722.037,A -85,B 0,C 180,E1 16427.753,E2 16427.753} C_VEL
LIN {X 0,Y 391.506,Z 705.14,A -85,B 0,C 180,E1 16426.81,E2 16426.81} C_VEL
LIN {X 0,Y 385.132,Z 688.256,A -85,B 0,C 180,E1 16424.504,E2 16424.504} C_VEL
LIN {X 0,Y 380.814,Z 669.856,A -85,B 0,C 180,E1 16422.131,E2 16422.131} C_VEL
LIN {X 0,Y 378.652,Z 649.962,A -85,B 0,C 180,E1 16419.718,E2 16419.718} C_VEL
LIN {X 0,Y 378.762,Z 629.275,A -85,B 0,C 180,E1 16417.384,E2 16417.384} C_VEL
LIN {X 0,Y 381.463,Z 603.88,A -85,B 0,C 180,E1 16414.744,E2 16414.744} C_VEL
LIN {X 0,Y 386.841,Z 573.241,A -85,B 0,C 180,E1 16411.77,E2 16411.77} C_VEL
LIN {X 0,Y 378.568,Z 554.851,A -85,B 0,C 180,E1 16408.214,E2 16408.214} C_VEL
LIN {X 0,Y 370.411,Z 537.678,A -85,B 0,C 180,E1 16404.542,E2 16404.542} C_VEL
LIN {X 0,Y 362.685,Z 521.784,A -85,B 0,C 180,E1 16400.832,E2 16400.832} C_VEL
LIN {X 0,Y 355.728,Z 508.154,A -85,B 0,C 180,E1 16397.334,E2 16397.334} C_VEL
LIN {X 0,Y 350.067,Z 496.774,A -85,B 0,C 180,E1 16394.219,E2 16394.219} C_VEL
LIN {X 0,Y 344.638,Z 486.773,A -85,B 0,C 180,E1 16391.208,E2 16391.208} C_VEL
LIN {X 0,Y 342.197,Z 482.15,A -85,B 0,C 180,E1 16389.757,E2 16389.757} C_VEL
LIN {X 0,Y 340.15,Z 477.944,A -85,B 0,C 180,E1 16388.451,E2 16388.451} C_VEL
LIN {X 0,Y 338.246,Z 474.587,A -85,B 0,C 180,E1 16387.302,E2 16387.302} C_VEL
LIN {X 0,Y 337.996,Z 473.382,A -85,B 0,C 180,E1 16386.966,E2 16386.966} C_VEL
LIN {X 0,Y 337.955,Z 473.386,A -85,B 0,C 180,E1 16382.713,E2 16382.713} C_VEL
LIN {X 0,Y 337.99,Z 473.38,A -85,B 0,C 180,E1 16378.474,E2 16378.474} C_VEL
LIN {X 0,Y 337.951,Z 473.387,A -85,B 0,C 180,E1 16374.226,E2 16374.226} C_VEL
LIN {X 0,Y 337.987,Z 473.382,A -85,B 0,C 180,E1 16369.948,E2 16369.948} C_VEL
LIN {X 0,Y 337.945,Z 473.373,A -85,B 0,C 180,E1 16365.609,E2 16365.609} C_VEL
LIN {X 0,Y 337.983,Z 473.361,A -85,B 0,C 180,E1 16361.367,E2 16361.367} C_VEL
LIN {X 0,Y 337.961,Z 473.366,A -85,B 0,C 180,E1 16356.828,E2 16356.828} C_VEL
LIN {X 0,Y 337.978,Z 473.367,A -85,B 0,C 180,E1 16352.706,E2 16352.706} C_VEL
LIN {X 0,Y 337.997,Z 473.622,A -85,B 0,C 180,E1 16351.256,E2 16351.256} C_VEL
LIN {X 0,Y 339.233,Z 476.813,A -85,B 0,C 180,E1 16350.397,E2 16350.397} C_VEL
LIN {X 0,Y 341.424,Z 479.465,A -85,B 0,C 180,E1 16349.365,E2 16349.365} C_VEL
LIN {X 0,Y 343.57,Z 483.314,A -85,B 0,C 180,E1 16348.214,E2 16348.214} C_VEL
LIN {X 0,Y 344.614,Z 484.745,A -85,B 0,C 180,E1 16347.733,E2 16347.733} C_VEL
LIN {X 0,Y 346.883,Z 488.677,A -85,B 0,C 180,E1 16346.596,E2 16346.596} C_VEL
LIN {X 0,Y 352.656,Z 498.933,A -85,B 0,C 180,E1 16343.862,E2 16343.862} C_VEL
LIN {X 0,Y 356.653,Z 506.259,A -85,B 0,C 180,E1 16342.174,E2 16342.174} C_VEL
LIN {X 0,Y 365.355,Z 518.89,A -85,B 0,C 180,E1 16340.052,E2 16340.052} C_VEL
LIN {X 0,Y 375.038,Z 534.226,A -85,B 0,C 180,E1 16337.868,E2 16337.868} C_VEL
LIN {X 0,Y 385.095,Z 551.952,A -85,B 0,C 180,E1 16335.756,E2 16335.756} C_VEL
LIN {X 0,Y 385.705,Z 553.458,A -85,B 0,C 180,E1 16335.622,E2 16335.622} C_VEL
LIN {X 0,Y 376.618,Z 765.69,A -85,B 0,C 180,E1 16331.436,E2 16331.436} C_VEL
LIN {X 0,Y 374.97,Z 786.159,A -85,B 0,C 180,E1 16330.789,E2 16330.789} C_VEL
LIN {X 0,Y 372.573,Z 806.695,A -85,B 0,C 180,E1 16329.867,E2 16329.867} C_VEL
LIN {X 0,Y 369.792,Z 825.493,A -85,B 0,C 180,E1 16328.75,E2 16328.75} C_VEL
LIN {X 0,Y 366.509,Z 843.92,A -85,B 0,C 180,E1 16327.371,E2 16327.371} C_VEL
LIN {X 0,Y 362.692,Z 862.259,A -85,B 0,C 180,E1 16325.665,E2 16325.665} C_VEL
LIN {X 0,Y 358.68,Z 879.496,A -85,B 0,C 180,E1 16323.691,E2 16323.691} C_VEL
LIN {X 0,Y 354.731,Z 895.132,A -85,B 0,C 180,E1 16321.523,E2 16321.523} C_VEL
LIN {X 0,Y 350.939,Z 909.385,A -85,B 0,C 180,E1 16319.155,E2 16319.155} C_VEL
LIN {X 0,Y 347.245,Z 923.035,A -85,B 0,C 180,E1 16316.427,E2 16316.427} C_VEL
LIN {X 0,Y 344.132,Z 934.642,A -85,B 0,C 180,E1 16313.637,E2 16313.637} C_VEL
LIN {X 0,Y 341.428,Z 945.155,A -85,B 0,C 180,E1 16310.573,E2 16310.573} C_VEL
LIN {X 0,Y 339.186,Z 954.61,A -85,B 0,C 180,E1 16307.143,E2 16307.143} C_VEL
LIN {X 0,Y 337.67,Z 962.031,A -85,B 0,C 180,E1 16303.702,E2 16303.702} C_VEL
LIN {X 0,Y 336.759,Z 967.629,A -85,B 0,C 180,E1 16300.261,E2 16300.261} C_VEL
LIN {X 0,Y 336.303,Z 971.598,A -85,B 0,C 180,E1 16296.775,E2 16296.775} C_VEL
LIN {X 0,Y 336.115,Z 973.901,A -85,B 0,C 180,E1 16293.41,E2 16293.41} C_VEL
LIN {X 0,Y 336.087,Z 974.722,A -85,B 0,C 180,E1 16289.999,E2 16289.999} C_VEL
LIN {X 0,Y 336.112,Z 973.939,A -85,B 0,C 180,E1 16286.588,E2 16286.588} C_VEL
LIN {X 0,Y 336.253,Z 972.144,A -85,B 0,C 180,E1 16283.732,E2 16283.732} C_VEL
LIN {X 0,Y 335.393,Z 971.061,A -85,B 0,C 180,E1 16282.431,E2 16282.431} C_VEL
LIN {X 0,Y 329.61,Z 967.32,A -85,B 0,C 180,E1 16278.853,E2 16278.853} C_VEL
LIN {X 0,Y 329.211,Z 965.783,A -85,B 0,C 180,E1 16277.822,E2 16277.822} C_VEL
LIN {X 0,Y 330.435,Z 959.562,A -85,B 0,C 180,E1 16274.376,E2 16274.376} C_VEL
LIN {X 0,Y 332.386,Z 951.209,A -85,B 0,C 180,E1 16270.831,E2 16270.831} C_VEL
LIN {X 0,Y 334.951,Z 941.427,A -85,B 0,C 180,E1 16267.536,E2 16267.536} C_VEL
LIN {X 0,Y 337.928,Z 930.742,A -85,B 0,C 180,E1 16264.593,E2 16264.593} C_VEL
LIN {X 0,Y 341.573,Z 918.008,A -85,B 0,C 180,E1 16261.691,E2 16261.691} C_VEL
LIN {X 0,Y 345.635,Z 903.733,A -85,B 0,C 180,E1 16259.007,E2 16259.007} C_VEL
LIN {X 0,Y 349.674,Z 888.978,A -85,B 0,C 180,E1 16256.7,E2 16256.7} C_VEL
LIN {X 0,Y 353.837,Z 872.764,A -85,B 0,C 180,E1 16254.599,E2 16254.599} C_VEL
LIN {X 0,Y 357.734,Z 855.899,A -85,B 0,C 180,E1 16252.804,E2 16252.804} C_VEL
LIN {X 0,Y 361.306,Z 838.54,A -85,B 0,C 180,E1 16251.286,E2 16251.286} C_VEL
LIN {X 0,Y 364.795,Z 818.763,A -85,B 0,C 180,E1 16249.9,E2 16249.9} C_VEL
LIN {X 0,Y 367.582,Z 799.079,A -85,B 0,C 180,E1 16248.831,E2 16248.831} C_VEL
LIN {X 0,Y 369.727,Z 779.042,A -85,B 0,C 180,E1 16248.024,E2 16248.024} C_VEL
LIN {X 0,Y 371.211,Z 757.714,A -85,B 0,C 180,E1 16247.449,E2 16247.449} C_VEL
LIN {X 0,Y 379.785,Z 561.868,A -85,B 0,C 180,E1 16243.565,E2 16243.565} C_VEL
LIN {X 0,Y 369.902,Z 543.636,A -85,B 0,C 180,E1 16241.394,E2 16241.394} C_VEL
LIN {X 0,Y 364.344,Z 534.399,A -85,B 0,C 180,E1 16240.107,E2 16240.107} C_VEL
LIN {X 0,Y 360.59,Z 535.38,A -85,B 0,C 180,E1 16239.419,E2 16239.419} C_VEL
LIN {X 0,Y 359.319,Z 535.49,A -85,B 0,C 180,E1 16239.173,E2 16239.173} C_VEL
LIN {X 0,Y 356.707,Z 536.63,A -85,B 0,C 180,E1 16238.688,E2 16238.688} C_VEL
LIN {X 0,Y 354.6,Z 536.008,A -85,B 0,C 180,E1 16238.238,E2 16238.238} C_VEL
LIN {X 0,Y 354.499,Z 536.086,A -85,B 0,C 180,E1 16238.148,E2 16238.148} C_VEL
LIN {X 0,Y 357.89,Z 547.047,A -85,B 0,C 180,E1 16236.121,E2 16236.121} C_VEL
LIN {X 0,Y 353.343,Z 581.238,A -85,B 0,C 180,E1 16231.853,E2 16231.853} C_VEL
LIN {X 0,Y 349.103,Z 617.043,A -85,B 0,C 180,E1 16227.459,E2 16227.459} C_VEL
LIN {X 0,Y 347.536,Z 633.003,A -85,B 0,C 180,E1 16225.575,E2 16225.575} C_VEL
LIN {X 0,Y 347.845,Z 639.098,A -85,B 0,C 180,E1 16225.325,E2 16225.325} C_VEL
LIN {X 0,Y 340.495,Z 765.081,A -85,B 0,C 180,E1 16221.173,E2 16221.173} C_VEL
LIN {X 0,Y 339.822,Z 784.707,A -85,B 0,C 180,E1 16220.361,E2 16220.361} C_VEL
LIN {X 0,Y 338.853,Z 802.074,A -85,B 0,C 180,E1 16219.298,E2 16219.298} C_VEL
LIN {X 0,Y 337.719,Z 817.572,A -85,B 0,C 180,E1 16218.022,E2 16218.022} C_VEL
LIN {X 0,Y 336.363,Z 832.958,A -85,B 0,C 180,E1 16216.403,E2 16216.403} C_VEL
LIN {X 0,Y 334.893,Z 847.659,A -85,B 0,C 180,E1 16214.436,E2 16214.436} C_VEL
LIN {X 0,Y 333.648,Z 859.543,A -85,B 0,C 180,E1 16212.461,E2 16212.461} C_VEL
LIN {X 0,Y 332.435,Z 871.301,A -85,B 0,C 180,E1 16210.047,E2 16210.047} C_VEL
LIN {X 0,Y 331.483,Z 881.224,A -85,B 0,C 180,E1 16207.453,E2 16207.453} C_VEL
LIN {X 0,Y 330.852,Z 889.026,A -85,B 0,C 180,E1 16204.854,E2 16204.854} C_VEL
LIN {X 0,Y 330.516,Z 895.317,A -85,B 0,C 180,E1 16202.081,E2 16202.081} C_VEL
LIN {X 0,Y 330.471,Z 899.726,A -85,B 0,C 180,E1 16199.307,E2 16199.307} C_VEL
LIN {X 0,Y 330.745,Z 902.562,A -85,B 0,C 180,E1 16196.36,E2 16196.36} C_VEL
LIN {X 0,Y 331.356,Z 903.476,A -85,B 0,C 180,E1 16193.416,E2 16193.416} C_VEL
LIN {X 0,Y 332.288,Z 902.637,A -85,B 0,C 180,E1 16190.649,E2 16190.649} C_VEL
LIN {X 0,Y 333.761,Z 899.953,A -85,B 0,C 180,E1 16187.72,E2 16187.72} C_VEL
LIN {X 0,Y 335.745,Z 895.242,A -85,B 0,C 180,E1 16184.808,E2 16184.808} C_VEL
LIN {X 0,Y 338.149,Z 888.85,A -85,B 0,C 180,E1 16182.091,E2 16182.091} C_VEL
LIN {X 0,Y 340.712,Z 881.491,A -85,B 0,C 180,E1 16179.74,E2 16179.74} C_VEL
LIN {X 0,Y 343.71,Z 872.196,A -85,B 0,C 180,E1 16177.419,E2 16177.419} C_VEL
LIN {X 0,Y 347.13,Z 860.489,A -85,B 0,C 180,E1 16175.132,E2 16175.132} C_VEL
LIN {X 0,Y 350.531,Z 847.391,A -85,B 0,C 180,E1 16173.121,E2 16173.121} C_VEL
LIN {X 0,Y 353.806,Z 833.016,A -85,B 0,C 180,E1 16171.38,E2 16171.38} C_VEL
LIN {X 0,Y 356.699,Z 818.418,A -85,B 0,C 180,E1 16169.977,E2 16169.977} C_VEL
LIN {X 0,Y 361.329,Z 794.474,A -85,B 0,C 180,E1 16168.187,E2 16168.187} C_VEL
LIN {X 0,Y 368.817,Z 765.375,A -85,B 0,C 180,E1 16166.34,E2 16166.34} C_VEL
LIN {X 0,Y 379.283,Z 727.106,A -85,B 0,C 180,E1 16164.367,E2 16164.367} C_VEL
LIN {X 0,Y 388.335,Z 690.553,A -85,B 0,C 180,E1 16162.767,E2 16162.767} C_VEL
LIN {X 0,Y 396.496,Z 679.503,A -85,B 0,C 180,E1 16162.038,E2 16162.038} C_VEL
LIN {X 0,Y 391.6,Z 689.364,A -85,B 0,C 180,E1 16159.761,E2 16159.761} C_VEL
LIN {X 0,Y 389.159,Z 699.428,A -85,B 0,C 180,E1 16157.401,E2 16157.401} C_VEL
LIN {X 0,Y 389.313,Z 709.983,A -85,B 0,C 180,E1 16154.934,E2 16154.934} C_VEL
LIN {X 0,Y 389.602,Z 711.713,A -85,B 0,C 180,E1 16154.534,E2 16154.534} C_VEL
LIN {X 0,Y 386.734,Z 717.559,A -85,B 0,C 180,E1 16154.253,E2 16154.253} C_VEL
LIN {X 0,Y 384.469,Z 728.398,A -85,B 0,C 180,E1 16153.997,E2 16153.997} C_VEL
LIN {X 0,Y 379.179,Z 750.472,A -85,B 0,C 180,E1 16153.706,E2 16153.706} C_VEL
LIN {X 0,Y 374.393,Z 769.495,A -85,B 0,C 180,E1 16153.238,E2 16153.238} C_VEL
LIN {X 0,Y 370.25,Z 786.199,A -85,B 0,C 180,E1 16152.57,E2 16152.57} C_VEL
LIN {X 0,Y 369.378,Z 790.939,A -85,B 0,C 180,E1 16152.369,E2 16152.369} C_VEL
LIN {X 0,Y 367.591,Z 812.1,A -85,B 0,C 180,E1 16151.779,E2 16151.779} C_VEL
LIN {X 0,Y 365.107,Z 831.816,A -85,B 0,C 180,E1 16150.987,E2 16150.987} C_VEL
LIN {X 0,Y 362.046,Z 850.984,A -85,B 0,C 180,E1 16149.949,E2 16149.949} C_VEL
LIN {X 0,Y 358.548,Z 869.413,A -85,B 0,C 180,E1 16148.658,E2 16148.658} C_VEL
LIN {X 0,Y 354.65,Z 887.561,A -85,B 0,C 180,E1 16147.074,E2 16147.074} C_VEL
LIN {X 0,Y 350.298,Z 905.818,A -85,B 0,C 180,E1 16145.111,E2 16145.111} C_VEL
LIN {X 0,Y 346.228,Z 921.873,A -85,B 0,C 180,E1 16143.006,E2 16143.006} C_VEL
LIN {X 0,Y 342.164,Z 937.348,A -85,B 0,C 180,E1 16140.562,E2 16140.562} C_VEL
LIN {X 0,Y 338.36,Z 951.665,A -85,B 0,C 180,E1 16137.834,E2 16137.834} C_VEL
LIN {X 0,Y 335.063,Z 964.446,A -85,B 0,C 180,E1 16134.883,E2 16134.883} C_VEL
LIN {X 0,Y 332.517,Z 975.193,A -85,B 0,C 180,E1 16131.893,E2 16131.893} C_VEL
LIN {X 0,Y 330.431,Z 985.154,A -85,B 0,C 180,E1 16128.526,E2 16128.526} C_VEL
LIN {X 0,Y 329.114,Z 993.192,A -85,B 0,C 180,E1 16125.146,E2 16125.146} C_VEL
LIN {X 0,Y 328.422,Z 999.505,A -85,B 0,C 180,E1 16121.771,E2 16121.771} C_VEL
LIN {X 0,Y 328.176,Z 1004.306,A -85,B 0,C 180,E1 16118.234,E2 16118.234} C_VEL
LIN {X 0,Y 328.175,Z 1007.254,A -85,B 0,C 180,E1 16114.895,E2 16114.895} C_VEL
LIN {X 0,Y 328.254,Z 1008.736,A -85,B 0,C 180,E1 16111.572,E2 16111.572} C_VEL
LIN {X 0,Y 328.255,Z 1008.759,A -85,B 0,C 180,E1 16108.605,E2 16108.605} C_VEL
LIN {X 0,Y 328.178,Z 1007.366,A -85,B 0,C 180,E1 16105.282,E2 16105.282} C_VEL
LIN {X 0,Y 328.15,Z 1004.51,A -85,B 0,C 180,E1 16101.944,E2 16101.944} C_VEL
LIN {X 0,Y 328.378,Z 999.762,A -85,B 0,C 180,E1 16098.408,E2 16098.408} C_VEL
LIN {X 0,Y 329.039,Z 993.544,A -85,B 0,C 180,E1 16095.032,E2 16095.032} C_VEL
LIN {X 0,Y 330.313,Z 985.604,A -85,B 0,C 180,E1 16091.652,E2 16091.652} C_VEL
LIN {X 0,Y 332.347,Z 975.749,A -85,B 0,C 180,E1 16088.283,E2 16088.283} C_VEL
LIN {X 0,Y 334.996,Z 964.512,A -85,B 0,C 180,E1 16085.14,E2 16085.14} C_VEL
LIN {X 0,Y 338.311,Z 951.619,A -85,B 0,C 180,E1 16082.164,E2 16082.164} C_VEL
LIN {X 0,Y 342.24,Z 936.82,A -85,B 0,C 180,E1 16079.35,E2 16079.35} C_VEL
LIN {X 0,Y 346.287,Z 921.378,A -85,B 0,C 180,E1 16076.928,E2 16076.928} C_VEL
LIN {X 0,Y 350.409,Z 905.057,A -85,B 0,C 180,E1 16074.804,E2 16074.804} C_VEL
LIN {X 0,Y 354.637,Z 887.16,A -85,B 0,C 180,E1 16072.891,E2 16072.891} C_VEL
LIN {X 0,Y 358.68,Z 868.254,A -85,B 0,C 180,E1 16071.259,E2 16071.259} C_VEL
LIN {X 0,Y 362.188,Z 849.505,A -85,B 0,C 180,E1 16069.969,E2 16069.969} C_VEL
LIN {X 0,Y 365.299,Z 829.757,A -85,B 0,C 180,E1 16068.917,E2 16068.917} C_VEL
LIN {X 0,Y 367.891,Z 808.525,A -85,B 0,C 180,E1 16068.101,E2 16068.101} C_VEL
LIN {X 0,Y 369.514,Z 786.532,A -85,B 0,C 180,E1 16067.531,E2 16067.531} C_VEL
LIN {X 0,Y 371.035,Z 763.805,A -85,B 0,C 180,E1 16067.16,E2 16067.16} C_VEL
LIN {X 0,Y 374.406,Z 736.304,A -85,B 0,C 180,E1 16066.934,E2 16066.934} C_VEL
LIN {X 0,Y 377.699,Z 718.368,A -85,B 0,C 180,E1 16066.924,E2 16066.924} C_VEL
LIN {X 0,Y 383.528,Z 706.463,A -85,B 0,C 180,E1 16066.231,E2 16066.231} C_VEL
LIN {X 0,Y 377.446,Z 689.121,A -85,B 0,C 180,E1 16063.856,E2 16063.856} C_VEL
LIN {X 0,Y 373.45,Z 670.197,A -85,B 0,C 180,E1 16061.399,E2 16061.399} C_VEL
LIN {X 0,Y 371.67,Z 649.903,A -85,B 0,C 180,E1 16058.924,E2 16058.924} C_VEL
LIN {X 0,Y 372.275,Z 627.718,A -85,B 0,C 180,E1 16056.41,E2 16056.41} C_VEL
LIN {X 0,Y 375.399,Z 602.606,A -85,B 0,C 180,E1 16053.8,E2 16053.8} C_VEL
LIN {X 0,Y 380.179,Z 576.809,A -85,B 0,C 180,E1 16051.271,E2 16051.271} C_VEL
LIN {X 0,Y 371.733,Z 558.012,A -85,B 0,C 180,E1 16047.557,E2 16047.557} C_VEL
LIN {X 0,Y 363.347,Z 540.237,A -85,B 0,C 180,E1 16043.688,E2 16043.688} C_VEL
LIN {X 0,Y 355.32,Z 523.763,A -85,B 0,C 180,E1 16039.735,E2 16039.735} C_VEL
LIN {X 0,Y 346.773,Z 506.759,A -85,B 0,C 180,E1 16035.211,E2 16035.211} C_VEL
LIN {X 0,Y 341.287,Z 496.459,A -85,B 0,C 180,E1 16032.177,E2 16032.177} C_VEL
LIN {X 0,Y 336.9,Z 488.038,A -85,B 0,C 180,E1 16029.567,E2 16029.567} C_VEL
LIN {X 0,Y 334.52,Z 483.447,A -85,B 0,C 180,E1 16028.075,E2 16028.075} C_VEL
LIN {X 0,Y 332.716,Z 479.876,A -85,B 0,C 180,E1 16026.904,E2 16026.904} C_VEL
LIN {X 0,Y 330.292,Z 475.593,A -85,B 0,C 180,E1 16025.384,E2 16025.384} C_VEL
LIN {X 0,Y 330.047,Z 474.372,A -85,B 0,C 180,E1 16025.04,E2 16025.04} C_VEL
LIN {X 0,Y 330.036,Z 474.371,A -85,B 0,C 180,E1 16020.52,E2 16020.52} C_VEL
LIN {X 0,Y 330.029,Z 474.372,A -85,B 0,C 180,E1 16016.352,E2 16016.352} C_VEL
LIN {X 0,Y 330.035,Z 474.345,A -85,B 0,C 180,E1 16011.814,E2 16011.814} C_VEL
LIN {X 0,Y 330.011,Z 474.353,A -85,B 0,C 180,E1 16007.578,E2 16007.578} C_VEL
LIN {X 0,Y 330.046,Z 474.357,A -85,B 0,C 180,E1 16003.194,E2 16003.194} C_VEL
LIN {X 0,Y 330.015,Z 474.369,A -85,B 0,C 180,E1 15998.866,E2 15998.866} C_VEL
LIN {X 0,Y 330.054,Z 474.368,A -85,B 0,C 180,E1 15994.52,E2 15994.52} C_VEL
LIN {X 0,Y 330.055,Z 474.39,A -85,B 0,C 180,E1 15993.725,E2 15993.725} C_VEL
LIN {X 0,Y 331.092,Z 477.434,A -85,B 0,C 180,E1 15992.87,E2 15992.87} C_VEL
LIN {X 0,Y 333.651,Z 480.485,A -85,B 0,C 180,E1 15991.544,E2 15991.544} C_VEL
LIN {X 0,Y 335.287,Z 483.801,A -85,B 0,C 180,E1 15990.525,E2 15990.525} C_VEL
LIN {X 0,Y 336.998,Z 485.931,A -85,B 0,C 180,E1 15989.697,E2 15989.697} C_VEL
LIN {X 0,Y 339.438,Z 490.105,A -85,B 0,C 180,E1 15988.377,E2 15988.377} C_VEL
LIN {X 0,Y 343.627,Z 497.484,A -85,B 0,C 180,E1 15986.237,E2 15986.237} C_VEL
LIN {X 0,Y 348.263,Z 505.724,A -85,B 0,C 180,E1 15984.057,E2 15984.057} C_VEL
LIN {X 0,Y 358.037,Z 519.754,A -85,B 0,C 180,E1 15981.457,E2 15981.457} C_VEL
LIN {X 0,Y 367.377,Z 534.26,A -85,B 0,C 180,E1 15979.217,E2 15979.217} C_VEL
LIN {X 0,Y 377.528,Z 551.666,A -85,B 0,C 180,E1 15976.966,E2 15976.966} C_VEL
LIN {X 0,Y 380.02,Z 556.691,A -85,B 0,C 180,E1 15976.426,E2 15976.426} C_VEL
LIN {X 0,Y 370.657,Z 766.115,A -85,B 0,C 180,E1 15972.252,E2 15972.252} C_VEL
LIN {X 0,Y 368.951,Z 786.522,A -85,B 0,C 180,E1 15971.601,E2 15971.601} C_VEL
LIN {X 0,Y 366.454,Z 807.142,A -85,B 0,C 180,E1 15970.666,E2 15970.666} C_VEL
LIN {X 0,Y 363.573,Z 825.884,A -85,B 0,C 180,E1 15969.541,E2 15969.541} C_VEL
LIN {X 0,Y 360.157,Z 844.318,A -85,B 0,C 180,E1 15968.147,E2 15968.147} C_VEL
LIN {X 0,Y 356.259,Z 862.31,A -85,B 0,C 180,E1 15966.455,E2 15966.455} C_VEL
LIN {X 0,Y 352.15,Z 879.252,A -85,B 0,C 180,E1 15964.501,E2 15964.501} C_VEL
LIN {X 0,Y 348.007,Z 895.001,A -85,B 0,C 180,E1 15962.302,E2 15962.302} C_VEL
LIN {X 0,Y 343.882,Z 909.798,A -85,B 0,C 180,E1 15959.813,E2 15959.813} C_VEL
LIN {X 0,Y 340.093,Z 923.13,A -85,B 0,C 180,E1 15957.109,E2 15957.109} C_VEL
LIN {X 0,Y 336.706,Z 935.058,A -85,B 0,C 180,E1 15954.191,E2 15954.191} C_VEL
LIN {X 0,Y 333.837,Z 945.573,A -85,B 0,C 180,E1 15951.063,E2 15951.063} C_VEL
LIN {X 0,Y 331.447,Z 955.027,A -85,B 0,C 180,E1 15947.557,E2 15947.557} C_VEL
LIN {X 0,Y 329.818,Z 962.447,A -85,B 0,C 180,E1 15944.035,E2 15944.035} C_VEL
LIN {X 0,Y 328.834,Z 968.044,A -85,B 0,C 180,E1 15940.511,E2 15940.511} C_VEL
LIN {X 0,Y 328.33,Z 972.052,A -85,B 0,C 180,E1 15936.894,E2 15936.894} C_VEL
LIN {X 0,Y 328.123,Z 974.378,A -85,B 0,C 180,E1 15933.318,E2 15933.318} C_VEL
LIN {X 0,Y 328.099,Z 975.134,A -85,B 0,C 180,E1 15929.999,E2 15929.999} C_VEL
LIN {X 0,Y 328.127,Z 974.351,A -85,B 0,C 180,E1 15926.505,E2 15926.505} C_VEL
LIN {X 0,Y 328.332,Z 972.051,A -85,B 0,C 180,E1 15923.002,E2 15923.002} C_VEL
LIN {X 0,Y 328.817,Z 968.179,A -85,B 0,C 180,E1 15919.487,E2 15919.487} C_VEL
LIN {X 0,Y 329.211,Z 965.783,A -85,B 0,C 180,E1 15917.822,E2 15917.822} C_VEL
LIN {X 0,Y 328.599,Z 963.757,A -85,B 0,C 180,E1 15916.522,E2 15916.522} C_VEL
LIN {X 0,Y 323.87,Z 957.901,A -85,B 0,C 180,E1 15913.024,E2 15913.024} C_VEL
LIN {X 0,Y 323.725,Z 955.48,A -85,B 0,C 180,E1 15911.924,E2 15911.924} C_VEL
LIN {X 0,Y 326.206,Z 946.271,A -85,B 0,C 180,E1 15908.418,E2 15908.418} C_VEL
LIN {X 0,Y 329.424,Z 935.187,A -85,B 0,C 180,E1 15905.045,E2 15905.045} C_VEL
LIN {X 0,Y 333.029,Z 923.192,A -85,B 0,C 180,E1 15902.071,E2 15902.071} C_VEL
LIN {X 0,Y 337.04,Z 909.784,A -85,B 0,C 180,E1 15899.318,E2 15899.318} C_VEL
LIN {X 0,Y 341.381,Z 894.896,A -85,B 0,C 180,E1 15896.79,E2 15896.79} C_VEL
LIN {X 0,Y 345.736,Z 879.031,A -85,B 0,C 180,E1 15894.56,E2 15894.56} C_VEL
LIN {X 0,Y 349.979,Z 862.218,A -85,B 0,C 180,E1 15892.609,E2 15892.609} C_VEL
LIN {X 0,Y 354.111,Z 843.818,A -85,B 0,C 180,E1 15890.87,E2 15890.87} C_VEL
LIN {X 0,Y 357.893,Z 824.095,A -85,B 0,C 180,E1 15889.386,E2 15889.386} C_VEL
LIN {X 0,Y 360.977,Z 804.208,A -85,B 0,C 180,E1 15888.228,E2 15888.228} C_VEL
LIN {X 0,Y 363.332,Z 784.391,A -85,B 0,C 180,E1 15887.365,E2 15887.365} C_VEL
LIN {X 0,Y 365.013,Z 763.536,A -85,B 0,C 180,E1 15886.731,E2 15886.731} C_VEL
LIN {X 0,Y 374.125,Z 564.974,A -85,B 0,C 180,E1 15882.726,E2 15882.726} C_VEL
LIN {X 0,Y 364.653,Z 547.515,A -85,B 0,C 180,E1 15880.558,E2 15880.558} C_VEL
LIN {X 0,Y 361.924,Z 543.105,A -85,B 0,C 180,E1 15879.913,E2 15879.913} C_VEL
LIN {X 0,Y 359.171,Z 543.658,A -85,B 0,C 180,E1 15879.398,E2 15879.398} C_VEL
LIN {X 0,Y 355.946,Z 544.57,A -85,B 0,C 180,E1 15878.786,E2 15878.786} C_VEL
LIN {X 0,Y 354.371,Z 544.786,A -85,B 0,C 180,E1 15878.473,E2 15878.473} C_VEL
LIN {X 0,Y 352.103,Z 545.936,A -85,B 0,C 180,E1 15878.04,E2 15878.04} C_VEL
LIN {X 0,Y 349.993,Z 545.679,A -85,B 0,C 180,E1 15877.584,E2 15877.584} C_VEL
LIN {X 0,Y 349.515,Z 545.4,A -85,B 0,C 180,E1 15877.438,E2 15877.438} C_VEL
LIN {X 0,Y 350.855,Z 550.186,A -85,B 0,C 180,E1 15876.556,E2 15876.556} C_VEL
LIN {X 0,Y 346.041,Z 585.334,A -85,B 0,C 180,E1 15872.118,E2 15872.118} C_VEL
LIN {X 0,Y 341.549,Z 622.112,A -85,B 0,C 180,E1 15867.551,E2 15867.551} C_VEL
LIN {X 0,Y 340.323,Z 633.977,A -85,B 0,C 180,E1 15866.137,E2 15866.137} C_VEL
LIN {X 0,Y 340.597,Z 640.154,A -85,B 0,C 180,E1 15865.88,E2 15865.88} C_VEL
LIN {X 0,Y 333.08,Z 760.852,A -85,B 0,C 180,E1 15861.772,E2 15861.772} C_VEL
LIN {X 0,Y 332.23,Z 784.537,A -85,B 0,C 180,E1 15860.801,E2 15860.801} C_VEL
LIN {X 0,Y 331.267,Z 801.601,A -85,B 0,C 180,E1 15859.758,E2 15859.758} C_VEL
LIN {X 0,Y 330.091,Z 817.508,A -85,B 0,C 180,E1 15858.454,E2 15858.454} C_VEL
LIN {X 0,Y 328.678,Z 833.114,A -85,B 0,C 180,E1 15856.798,E2 15856.798} C_VEL
LIN {X 0,Y 327.274,Z 846.827,A -85,B 0,C 180,E1 15854.961,E2 15854.961} C_VEL
LIN {X 0,Y 325.952,Z 859.092,A -85,B 0,C 180,E1 15852.94,E2 15852.94} C_VEL
LIN {X 0,Y 324.739,Z 870.353,A -85,B 0,C 180,E1 15850.646,E2 15850.646} C_VEL
LIN {X 0,Y 323.76,Z 880.2,A -85,B 0,C 180,E1 15848.167,E2 15848.167} C_VEL
LIN {X 0,Y 323.009,Z 889.013,A -85,B 0,C 180,E1 15845.329,E2 15845.329} C_VEL
LIN {X 0,Y 322.627,Z 895.325,A -85,B 0,C 180,E1 15842.665,E2 15842.665} C_VEL
LIN {X 0,Y 322.548,Z 900.472,A -85,B 0,C 180,E1 15839.645,E2 15839.645} C_VEL
LIN {X 0,Y 322.808,Z 903.63,A -85,B 0,C 180,E1 15836.626,E2 15836.626} C_VEL
LIN {X 0,Y 323.383,Z 904.907,A -85,B 0,C 180,E1 15833.788,E2 15833.788} C_VEL
LIN {X 0,Y 324.472,Z 904.38,A -85,B 0,C 180,E1 15830.601,E2 15830.601} C_VEL
LIN {X 0,Y 326.02,Z 901.931,A -85,B 0,C 180,E1 15827.604,E2 15827.604} C_VEL
LIN {X 0,Y 327.989,Z 897.881,A -85,B 0,C 180,E1 15824.802,E2 15824.802} C_VEL
LIN {X 0,Y 330.5,Z 891.993,A -85,B 0,C 180,E1 15822.027,E2 15822.027} C_VEL
LIN {X 0,Y 333.716,Z 883.724,A -85,B 0,C 180,E1 15819.197,E2 15819.197} C_VEL
LIN {X 0,Y 337.287,Z 873.594,A -85,B 0,C 180,E1 15816.595,E2 15816.595} C_VEL
LIN {X 0,Y 340.988,Z 861.974,A -85,B 0,C 180,E1 15814.28,E2 15814.28} C_VEL
LIN {X 0,Y 344.532,Z 849.668,A -85,B 0,C 180,E1 15812.333,E2 15812.333} C_VEL
LIN {X 0,Y 348.099,Z 835.854,A -85,B 0,C 180,E1 15810.583,E2 15810.583} C_VEL
LIN {X 0,Y 351.622,Z 820.307,A -85,B 0,C 180,E1 15809.024,E2 15809.024} C_VEL
LIN {X 0,Y 356.984,Z 796.886,A -85,B 0,C 180,E1 15807.183,E2 15807.183} C_VEL
LIN {X 0,Y 364.978,Z 769.327,A -85,B 0,C 180,E1 15805.358,E2 15805.358} C_VEL
LIN {X 0,Y 375.23,Z 735.349,A -85,B 0,C 180,E1 15803.543,E2 15803.543} C_VEL
LIN {X 0,Y 385.799,Z 695.561,A -85,B 0,C 180,E1 15801.775,E2 15801.775} C_VEL
LIN {X 0,Y 386.374,Z 693.857,A -85,B 0,C 180,E1 15801.7,E2 15801.7} C_VEL
LIN {X 0,Y 389.333,Z 689.935,A -85,B 0,C 180,E1 15801.472,E2 15801.472} C_VEL
LIN {X 0,Y 385.205,Z 699.963,A -85,B 0,C 180,E1 15799.056,E2 15799.056} C_VEL
LIN {X 0,Y 383.727,Z 709.845,A -85,B 0,C 180,E1 15796.655,E2 15796.655} C_VEL
LIN {X 0,Y 384.382,Z 715.646,A -85,B 0,C 180,E1 15795.432,E2 15795.432} C_VEL
LIN {X 0,Y 381.6,Z 728.322,A -85,B 0,C 180,E1 15795.115,E2 15795.115} C_VEL
LIN {X 0,Y 376.016,Z 750.306,A -85,B 0,C 180,E1 15794.823,E2 15794.823} C_VEL
LIN {X 0,Y 370.849,Z 769.337,A -85,B 0,C 180,E1 15794.346,E2 15794.346} C_VEL
LIN {X 0,Y 366.235,Z 786.237,A -85,B 0,C 180,E1 15793.658,E2 15793.658} C_VEL
LIN {X 0,Y 362.856,Z 799.443,A -85,B 0,C 180,E1 15793.001,E2 15793.001} C_VEL
LIN {X 0,Y 360.71,Z 819.748,A -85,B 0,C 180,E1 15792.338,E2 15792.338} C_VEL
LIN {X 0,Y 357.676,Z 840.291,A -85,B 0,C 180,E1 15791.386,E2 15791.386} C_VEL
LIN {X 0,Y 354.137,Z 859.74,A -85,B 0,C 180,E1 15790.177,E2 15790.177} C_VEL
LIN {X 0,Y 350.221,Z 878.367,A -85,B 0,C 180,E1 15788.7,E2 15788.7} C_VEL
LIN {X 0,Y 346.003,Z 896.213,A -85,B 0,C 180,E1 15786.947,E2 15786.947} C_VEL
LIN {X 0,Y 341.588,Z 913.222,A -85,B 0,C 180,E1 15784.908,E2 15784.908} C_VEL
LIN {X 0,Y 337.233,Z 929.32,A -85,B 0,C 180,E1 15782.557,E2 15782.557} C_VEL
LIN {X 0,Y 333.003,Z 944.396,A -85,B 0,C 180,E1 15779.897,E2 15779.897} C_VEL
LIN {X 0,Y 329.162,Z 958.307,A -85,B 0,C 180,E1 15776.912,E2 15776.912} C_VEL
LIN {X 0,Y 325.911,Z 970.603,A -85,B 0,C 180,E1 15773.698,E2 15773.698} C_VEL
LIN {X 0,Y 323.47,Z 980.798,A -85,B 0,C 180,E1 15770.445,E2 15770.445} C_VEL
LIN {X 0,Y 321.747,Z 989.604,A -85,B 0,C 180,E1 15766.986,E2 15766.986} C_VEL
LIN {X 0,Y 320.678,Z 996.919,A -85,B 0,C 180,E1 15763.341,E2 15763.341} C_VEL
LIN {X 0,Y 320.235,Z 1002.178,A -85,B 0,C 180,E1 15759.889,E2 15759.889} C_VEL
LIN {X 0,Y 320.168,Z 1005.8,A -85,B 0,C 180,E1 15756.456,E2 15756.456} C_VEL
LIN {X 0,Y 320.23,Z 1007.87,A -85,B 0,C 180,E1 15753.044,E2 15753.044} C_VEL
LIN {X 0,Y 320.275,Z 1008.488,A -85,B 0,C 180,E1 15749.643,E2 15749.643} C_VEL
LIN {X 0,Y 320.215,Z 1007.653,A -85,B 0,C 180,E1 15746.421,E2 15746.421} C_VEL
LIN {X 0,Y 320.133,Z 1005.294,A -85,B 0,C 180,E1 15743.005,E2 15743.005} C_VEL
LIN {X 0,Y 320.261,Z 1001.425,A -85,B 0,C 180,E1 15739.554,E2 15739.554} C_VEL
LIN {X 0,Y 320.807,Z 995.654,A -85,B 0,C 180,E1 15735.931,E2 15735.931} C_VEL
LIN {X 0,Y 322.021,Z 987.922,A -85,B 0,C 180,E1 15732.286,E2 15732.286} C_VEL
LIN {X 0,Y 323.924,Z 978.666,A -85,B 0,C 180,E1 15728.831,E2 15728.831} C_VEL
LIN {X 0,Y 326.503,Z 967.977,A -85,B 0,C 180,E1 15725.582,E2 15725.582} C_VEL
LIN {X 0,Y 329.944,Z 955.133,A -85,B 0,C 180,E1 15722.378,E2 15722.378} C_VEL
LIN {X 0,Y 333.709,Z 941.56,A -85,B 0,C 180,E1 15719.58,E2 15719.58} C_VEL
LIN {X 0,Y 337.92,Z 926.566,A -85,B 0,C 180,E1 15717.015,E2 15717.015} C_VEL
LIN {X 0,Y 342.375,Z 910.023,A -85,B 0,C 180,E1 15714.675,E2 15714.675} C_VEL
LIN {X 0,Y 346.865,Z 892.408,A -85,B 0,C 180,E1 15712.644,E2 15712.644} C_VEL
LIN {X 0,Y 351.156,Z 873.709,A -85,B 0,C 180,E1 15710.9,E2 15710.9} C_VEL
LIN {X 0,Y 354.891,Z 855.251,A -85,B 0,C 180,E1 15709.525,E2 15709.525} C_VEL
LIN {X 0,Y 358.297,Z 835.635,A -85,B 0,C 180,E1 15708.383,E2 15708.383} C_VEL
LIN {X 0,Y 361.116,Z 815.302,A -85,B 0,C 180,E1 15707.501,E2 15707.501} C_VEL
LIN {X 0,Y 363.12,Z 794.686,A -85,B 0,C 180,E1 15706.874,E2 15706.874} C_VEL
LIN {X 0,Y 364.679,Z 769.379,A -85,B 0,C 180,E1 15706.383,E2 15706.383} C_VEL
LIN {X 0,Y 368.115,Z 739.191,A -85,B 0,C 180,E1 15706.096,E2 15706.096} C_VEL
LIN {X 0,Y 372.528,Z 714.55,A -85,B 0,C 180,E1 15706.069,E2 15706.069} C_VEL
LIN {X 0,Y 375.792,Z 708.192,A -85,B 0,C 180,E1 15705.702,E2 15705.702} C_VEL
LIN {X 0,Y 369.946,Z 690.397,A -85,B 0,C 180,E1 15703.246,E2 15703.246} C_VEL
LIN {X 0,Y 366.231,Z 671.141,A -85,B 0,C 180,E1 15700.73,E2 15700.73} C_VEL
LIN {X 0,Y 364.774,Z 650.336,A -85,B 0,C 180,E1 15698.167,E2 15698.167} C_VEL
LIN {X 0,Y 365.704,Z 627.914,A -85,B 0,C 180,E1 15695.616,E2 15695.616} C_VEL
LIN {X 0,Y 369.254,Z 602.181,A -85,B 0,C 180,E1 15692.923,E2 15692.923} C_VEL
LIN {X 0,Y 373.483,Z 580.331,A -85,B 0,C 180,E1 15690.752,E2 15690.752} C_VEL
LIN {X 0,Y 365.174,Z 561.782,A -85,B 0,C 180,E1 15687.033,E2 15687.033} C_VEL
LIN {X 0,Y 356.804,Z 544.08,A -85,B 0,C 180,E1 15683.098,E2 15683.098} C_VEL
LIN {X 0,Y 349.44,Z 528.808,A -85,B 0,C 180,E1 15679.385,E2 15679.385} C_VEL
LIN {X 0,Y 341.18,Z 512.27,A -85,B 0,C 180,E1 15674.945,E2 15674.945} C_VEL
LIN {X 0,Y 334.417,Z 499.1,A -85,B 0,C 180,E1 15671.031,E2 15671.031} C_VEL
LIN {X 0,Y 328.863,Z 488.845,A -85,B 0,C 180,E1 15667.688,E2 15667.688} C_VEL
LIN {X 0,Y 326.834,Z 484.74,A -85,B 0,C 180,E1 15666.323,E2 15666.323} C_VEL
LIN {X 0,Y 324.941,Z 481.397,A -85,B 0,C 180,E1 15665.119,E2 15665.119} C_VEL
LIN {X 0,Y 324.222,Z 479.878,A -85,B 0,C 180,E1 15664.599,E2 15664.599} C_VEL
LIN {X 0,Y 322.339,Z 476.617,A -85,B 0,C 180,E1 15663.378,E2 15663.378} C_VEL
LIN {X 0,Y 322.085,Z 475.362,A -85,B 0,C 180,E1 15663.025,E2 15663.025} C_VEL
LIN {X 0,Y 322.115,Z 475.358,A -85,B 0,C 180,E1 15658.755,E2 15658.755} C_VEL
LIN {X 0,Y 322.075,Z 475.364,A -85,B 0,C 180,E1 15654.298,E2 15654.298} C_VEL
LIN {X 0,Y 322.11,Z 475.358,A -85,B 0,C 180,E1 15649.989,E2 15649.989} C_VEL
LIN {X 0,Y 322.072,Z 475.351,A -85,B 0,C 180,E1 15645.436,E2 15645.436} C_VEL
LIN {X 0,Y 322.101,Z 475.34,A -85,B 0,C 180,E1 15641.165,E2 15641.165} C_VEL
LIN {X 0,Y 322.112,Z 475.426,A -85,B 0,C 180,E1 15636.523,E2 15636.523} C_VEL
LIN {X 0,Y 323.233,Z 478.586,A -85,B 0,C 180,E1 15635.512,E2 15635.512} C_VEL
LIN {X 0,Y 325.949,Z 481.528,A -85,B 0,C 180,E1 15633.981,E2 15633.981} C_VEL
LIN {X 0,Y 327.718,Z 485.124,A -85,B 0,C 180,E1 15632.764,E2 15632.764} C_VEL
LIN {X 0,Y 329.34,Z 486.91,A -85,B 0,C 180,E1 15631.928,E2 15631.928} C_VEL
LIN {X 0,Y 331.247,Z 490.615,A -85,B 0,C 180,E1 15630.725,E2 15630.725} C_VEL
LIN {X 0,Y 332.799,Z 492.842,A -85,B 0,C 180,E1 15629.911,E2 15629.911} C_VEL
LIN {X 0,Y 336.253,Z 498.797,A -85,B 0,C 180,E1 15628.042,E2 15628.042} C_VEL
LIN {X 0,Y 340.948,Z 506.801,A -85,B 0,C 180,E1 15625.732,E2 15625.732} C_VEL
LIN {X 0,Y 351.245,Z 521.361,A -85,B 0,C 180,E1 15622.829,E2 15622.829} C_VEL
LIN {X 0,Y 360.185,Z 534.918,A -85,B 0,C 180,E1 15620.554,E2 15620.554} C_VEL
LIN {X 0,Y 370.199,Z 551.851,A -85,B 0,C 180,E1 15618.202,E2 15618.202} C_VEL
LIN {X 0,Y 374.412,Z 559.916,A -85,B 0,C 180,E1 15617.254,E2 15617.254} C_VEL
LIN {X 0,Y 364.771,Z 766.541,A -85,B 0,C 180,E1 15613.094,E2 15613.094} C_VEL
LIN {X 0,Y 362.997,Z 786.999,A -85,B 0,C 180,E1 15612.435,E2 15612.435} C_VEL
LIN {X 0,Y 360.414,Z 807.571,A -85,B 0,C 180,E1 15611.493,E2 15611.493} C_VEL
LIN {X 0,Y 357.426,Z 826.276,A -85,B 0,C 180,E1 15610.359,E2 15610.359} C_VEL
LIN {X 0,Y 353.872,Z 844.717,A -85,B 0,C 180,E1 15608.951,E2 15608.951} C_VEL
LIN {X 0,Y 349.76,Z 862.967,A -85,B 0,C 180,E1 15607.213,E2 15607.213} C_VEL
LIN {X 0,Y 345.531,Z 879.659,A -85,B 0,C 180,E1 15605.259,E2 15605.259} C_VEL
LIN {X 0,Y 341.198,Z 895.412,A -85,B 0,C 180,E1 15603.028,E2 15603.028} C_VEL
LIN {X 0,Y 336.876,Z 910.211,A -85,B 0,C 180,E1 15600.499,E2 15600.499} C_VEL
LIN {X 0,Y 332.892,Z 923.546,A -85,B 0,C 180,E1 15597.745,E2 15597.745} C_VEL
LIN {X 0,Y 329.312,Z 935.475,A -85,B 0,C 180,E1 15594.77,E2 15594.77} C_VEL
LIN {X 0,Y 326.27,Z 945.99,A -85,B 0,C 180,E1 15591.575,E2 15591.575} C_VEL
LIN {X 0,Y 323.723,Z 955.445,A -85,B 0,C 180,E1 15587.99,E2 15587.99} C_VEL
LIN {X 0,Y 321.978,Z 962.864,A -85,B 0,C 180,E1 15584.384,E2 15584.384} C_VEL
LIN {X 0,Y 320.915,Z 968.459,A -85,B 0,C 180,E1 15580.773,E2 15580.773} C_VEL
LIN {X 0,Y 320.371,Z 972.378,A -85,B 0,C 180,E1 15577.17,E2 15577.17} C_VEL
LIN {X 0,Y 320.145,Z 974.725,A -85,B 0,C 180,E1 15573.58,E2 15573.58} C_VEL
LIN {X 0,Y 320.105,Z 975.525,A -85,B 0,C 180,E1 15570.178,E2 15570.178} C_VEL
LIN {X 0,Y 320.13,Z 974.892,A -85,B 0,C 180,E1 15566.776,E2 15566.776} C_VEL
LIN {X 0,Y 320.334,Z 972.77,A -85,B 0,C 180,E1 15563.187,E2 15563.187} C_VEL
LIN {X 0,Y 320.823,Z 969.083,A -85,B 0,C 180,E1 15559.585,E2 15559.585} C_VEL
LIN {X 0,Y 321.814,Z 963.699,A -85,B 0,C 180,E1 15555.974,E2 15555.974} C_VEL
LIN {X 0,Y 323.468,Z 956.473,A -85,B 0,C 180,E1 15552.366,E2 15552.366} C_VEL
LIN {X 0,Y 323.725,Z 955.48,A -85,B 0,C 180,E1 15551.924,E2 15551.924} C_VEL
LIN {X 0,Y 323.521,Z 952.563,A -85,B 0,C 180,E1 15550.655,E2 15550.655} C_VEL
LIN {X 0,Y 320.078,Z 944.963,A -85,B 0,C 180,E1 15547.391,E2 15547.391} C_VEL
LIN {X 0,Y 320.266,Z 941.408,A -85,B 0,C 180,E1 15546.148,E2 15546.148} C_VEL
LIN {X 0,Y 323.774,Z 930.202,A -85,B 0,C 180,E1 15543.001,E2 15543.001} C_VEL
LIN {X 0,Y 327.644,Z 918.003,A -85,B 0,C 180,E1 15540.169,E2 15540.169} C_VEL
LIN {X 0,Y 332.145,Z 903.556,A -85,B 0,C 180,E1 15537.394,E2 15537.394} C_VEL
LIN {X 0,Y 336.784,Z 887.999,A -85,B 0,C 180,E1 15534.936,E2 15534.936} C_VEL
LIN {X 0,Y 341.184,Z 872.093,A -85,B 0,C 180,E1 15532.856,E2 15532.856} C_VEL
LIN {X 0,Y 345.465,Z 855.033,A -85,B 0,C 180,E1 15531.022,E2 15531.022} C_VEL
LIN {X 0,Y 349.548,Z 836.367,A -85,B 0,C 180,E1 15529.401,E2 15529.401} C_VEL
LIN {X 0,Y 352.989,Z 817.694,A -85,B 0,C 180,E1 15528.109,E2 15528.109} C_VEL
LIN {X 0,Y 355.987,Z 797.374,A -85,B 0,C 180,E1 15527.02,E2 15527.02} C_VEL
LIN {X 0,Y 358.301,Z 776.104,A -85,B 0,C 180,E1 15526.199,E2 15526.199} C_VEL
LIN {X 0,Y 359.838,Z 752.971,A -85,B 0,C 180,E1 15525.617,E2 15525.617} C_VEL
LIN {X 0,Y 368.559,Z 568.134,A -85,B 0,C 180,E1 15521.865,E2 15521.865} C_VEL
LIN {X 0,Y 359.541,Z 551.459,A -85,B 0,C 180,E1 15519.712,E2 15519.712} C_VEL
LIN {X 0,Y 354.205,Z 552.973,A -85,B 0,C 180,E1 15518.701,E2 15518.701} C_VEL
LIN {X 0,Y 350.712,Z 553.966,A -85,B 0,C 180,E1 15518.011,E2 15518.011} C_VEL
LIN {X 0,Y 349.463,Z 554.241,A -85,B 0,C 180,E1 15517.755,E2 15517.755} C_VEL
LIN {X 0,Y 344.927,Z 557.447,A -85,B 0,C 180,E1 15516.873,E2 15516.873} C_VEL
LIN {X 0,Y 343.195,Z 557.624,A -85,B 0,C 180,E1 15516.465,E2 15516.465} C_VEL
LIN {X 0,Y 338.409,Z 591.575,A -85,B 0,C 180,E1 15512.129,E2 15512.129} C_VEL
LIN {X 0,Y 333.927,Z 627.718,A -85,B 0,C 180,E1 15507.587,E2 15507.587} C_VEL
LIN {X 0,Y 333.159,Z 635.124,A -85,B 0,C 180,E1 15506.714,E2 15506.714} C_VEL
LIN {X 0,Y 333.38,Z 641.132,A -85,B 0,C 180,E1 15506.46,E2 15506.46} C_VEL
LIN {X 0,Y 325.43,Z 763.47,A -85,B 0,C 180,E1 15502.139,E2 15502.139} C_VEL
LIN {X 0,Y 324.562,Z 786.519,A -85,B 0,C 180,E1 15501.151,E2 15501.151} C_VEL
LIN {X 0,Y 323.53,Z 803.465,A -85,B 0,C 180,E1 15500.063,E2 15500.063} C_VEL
LIN {X 0,Y 322.31,Z 819.082,A -85,B 0,C 180,E1 15498.728,E2 15498.728} C_VEL
LIN {X 0,Y 320.85,Z 834.539,A -85,B 0,C 180,E1 15497.034,E2 15497.034} C_VEL
LIN {X 0,Y 319.431,Z 847.956,A -85,B 0,C 180,E1 15495.19,E2 15495.19} C_VEL
LIN {X 0,Y 318.051,Z 860.455,A -85,B 0,C 180,E1 15493.082,E2 15493.082} C_VEL
LIN {X 0,Y 316.811,Z 871.714,A -85,B 0,C 180,E1 15490.732,E2 15490.732} C_VEL
LIN {X 0,Y 315.813,Z 881.573,A -85,B 0,C 180,E1 15488.191,E2 15488.191} C_VEL
LIN {X 0,Y 315.055,Z 890.378,A -85,B 0,C 180,E1 15485.281,E2 15485.281} C_VEL
LIN {X 0,Y 314.674,Z 897.055,A -85,B 0,C 180,E1 15482.368,E2 15482.368} C_VEL
LIN {X 0,Y 314.633,Z 901.88,A -85,B 0,C 180,E1 15479.454,E2 15479.454} C_VEL
LIN {X 0,Y 314.943,Z 905.07,A -85,B 0,C 180,E1 15476.36,E2 15476.36} C_VEL
LIN {X 0,Y 315.599,Z 906.397,A -85,B 0,C 180,E1 15473.451,E2 15473.451} C_VEL
LIN {X 0,Y 316.726,Z 905.997,A -85,B 0,C 180,E1 15470.369,E2 15470.369} C_VEL
LIN {X 0,Y 318.399,Z 903.743,A -85,B 0,C 180,E1 15467.302,E2 15467.302} C_VEL
LIN {X 0,Y 320.519,Z 899.905,A -85,B 0,C 180,E1 15464.439,E2 15464.439} C_VEL
LIN {X 0,Y 323.404,Z 893.854,A -85,B 0,C 180,E1 15461.432,E2 15461.432} C_VEL
LIN {X 0,Y 326.748,Z 886.042,A -85,B 0,C 180,E1 15458.645,E2 15458.645} C_VEL
LIN {X 0,Y 330.443,Z 876.554,A -85,B 0,C 180,E1 15456.08,E2 15456.08} C_VEL
LIN {X 0,Y 334.404,Z 865.496,A -85,B 0,C 180,E1 15453.736,E2 15453.736} C_VEL
LIN {X 0,Y 338.688,Z 852.249,A -85,B 0,C 180,E1 15451.526,E2 15451.526} C_VEL
LIN {X 0,Y 342.9,Z 837.608,A -85,B 0,C 180,E1 15449.609,E2 15449.609} C_VEL
LIN {X 0,Y 346.991,Z 821.932,A -85,B 0,C 180,E1 15447.982,E2 15447.982} C_VEL
LIN {X 0,Y 353.16,Z 798.98,A -85,B 0,C 180,E1 15446.101,E2 15446.101} C_VEL
LIN {X 0,Y 362.018,Z 772.022,A -85,B 0,C 180,E1 15444.258,E2 15444.258} C_VEL
LIN {X 0,Y 372.396,Z 740.482,A -85,B 0,C 180,E1 15442.545,E2 15442.545} C_VEL
LIN {X 0,Y 381.818,Z 707.678,A -85,B 0,C 180,E1 15441.056,E2 15441.056} C_VEL
LIN {X 0,Y 383.544,Z 701.441,A -85,B 0,C 180,E1 15440.78,E2 15440.78} C_VEL
LIN {X 0,Y 381.238,Z 711.401,A -85,B 0,C 180,E1 15438.403,E2 15438.403} C_VEL
LIN {X 0,Y 381.211,Z 719.95,A -85,B 0,C 180,E1 15436.469,E2 15436.469} C_VEL
LIN {X 0,Y 379.091,Z 728.902,A -85,B 0,C 180,E1 15436.263,E2 15436.263} C_VEL
LIN {X 0,Y 373.35,Z 750.277,A -85,B 0,C 180,E1 15435.978,E2 15435.978} C_VEL
LIN {X 0,Y 367.501,Z 770.181,A -85,B 0,C 180,E1 15435.466,E2 15435.466} C_VEL
LIN {X 0,Y 362.63,Z 786.5,A -85,B 0,C 180,E1 15434.788,E2 15434.788} C_VEL
LIN {X 0,Y 356.158,Z 808.354,A -85,B 0,C 180,E1 15433.611,E2 15433.611} C_VEL
LIN {X 0,Y 353.344,Z 829.597,A -85,B 0,C 180,E1 15432.777,E2 15432.777} C_VEL
LIN {X 0,Y 350.036,Z 848.951,A -85,B 0,C 180,E1 15431.726,E2 15431.726} C_VEL
LIN {X 0,Y 346.249,Z 867.632,A -85,B 0,C 180,E1 15430.414,E2 15430.414} C_VEL
LIN {X 0,Y 341.869,Z 886.483,A -85,B 0,C 180,E1 15428.748,E2 15428.748} C_VEL
LIN {X 0,Y 337.252,Z 904.339,A -85,B 0,C 180,E1 15426.79,E2 15426.79} C_VEL
LIN {X 0,Y 332.725,Z 920.632,A -85,B 0,C 180,E1 15424.609,E2 15424.609} C_VEL
LIN {X 0,Y 328.356,Z 935.742,A -85,B 0,C 180,E1 15422.165,E2 15422.165} C_VEL
LIN {X 0,Y 323.875,Z 950.832,A -85,B 0,C 180,E1 15419.195,E2 15419.195} C_VEL
LIN {X 0,Y 320.183,Z 963.609,A -85,B 0,C 180,E1 15416.125,E2 15416.125} C_VEL
LIN {X 0,Y 317.128,Z 974.939,A -85,B 0,C 180,E1 15412.819,E2 15412.819} C_VEL
LIN {X 0,Y 314.78,Z 984.784,A -85,B 0,C 180,E1 15409.291,E2 15409.291} C_VEL
LIN {X 0,Y 313.221,Z 993.081,A -85,B 0,C 180,E1 15405.555,E2 15405.555} C_VEL
LIN {X 0,Y 312.424,Z 999.461,A -85,B 0,C 180,E1 15401.82,E2 15401.82} C_VEL
LIN {X 0,Y 312.181,Z 1003.931,A -85,B 0,C 180,E1 15398.244,E2 15398.244} C_VEL
LIN {X 0,Y 312.193,Z 1006.664,A -85,B 0,C 180,E1 15394.778,E2 15394.778} C_VEL
LIN {X 0,Y 312.277,Z 1007.961,A -85,B 0,C 180,E1 15391.285,E2 15391.285} C_VEL
LIN {X 0,Y 312.264,Z 1007.861,A -85,B 0,C 180,E1 15387.983,E2 15387.983} C_VEL
LIN {X 0,Y 312.166,Z 1006.184,A -85,B 0,C 180,E1 15384.487,E2 15384.487} C_VEL
LIN {X 0,Y 312.178,Z 1002.822,A -85,B 0,C 180,E1 15380.786,E2 15380.786} C_VEL
LIN {X 0,Y 312.533,Z 998.052,A -85,B 0,C 180,E1 15377.248,E2 15377.248} C_VEL
LIN {X 0,Y 313.515,Z 991.238,A -85,B 0,C 180,E1 15373.512,E2 15373.512} C_VEL
LIN {X 0,Y 315.28,Z 982.408,A -85,B 0,C 180,E1 15369.778,E2 15369.778} C_VEL
LIN {X 0,Y 317.684,Z 972.561,A -85,B 0,C 180,E1 15366.441,E2 15366.441} C_VEL
LIN {X 0,Y 320.727,Z 961.426,A -85,B 0,C 180,E1 15363.327,E2 15363.327} C_VEL
LIN {X 0,Y 324.56,Z 948.206,A -85,B 0,C 180,E1 15360.266,E2 15360.266} C_VEL
LIN {X 0,Y 328.836,Z 933.726,A -85,B 0,C 180,E1 15357.498,E2 15357.498} C_VEL
LIN {X 0,Y 333.332,Z 918.24,A -85,B 0,C 180,E1 15355.047,E2 15355.047} C_VEL
LIN {X 0,Y 338.12,Z 900.859,A -85,B 0,C 180,E1 15352.792,E2 15352.792} C_VEL
LIN {X 0,Y 342.822,Z 882.276,A -85,B 0,C 180,E1 15350.845,E2 15350.845} C_VEL
LIN {X 0,Y 347.072,Z 863.323,A -85,B 0,C 180,E1 15349.258,E2 15349.258} C_VEL
LIN {X 0,Y 350.647,Z 844.883,A -85,B 0,C 180,E1 15348.037,E2 15348.037} C_VEL
LIN {X 0,Y 353.992,Z 824.162,A -85,B 0,C 180,E1 15346.992,E2 15346.992} C_VEL
LIN {X 0,Y 356.572,Z 802.793,A -85,B 0,C 180,E1 15346.227,E2 15346.227} C_VEL
LIN {X 0,Y 358.151,Z 779.681,A -85,B 0,C 180,E1 15345.67,E2 15345.67} C_VEL
LIN {X 0,Y 360.384,Z 754.94,A -85,B 0,C 180,E1 15345.342,E2 15345.342} C_VEL
LIN {X 0,Y 363.565,Z 731.391,A -85,B 0,C 180,E1 15345.197,E2 15345.197} C_VEL
LIN {X 0,Y 367.472,Z 710.682,A -85,B 0,C 180,E1 15345.195,E2 15345.195} C_VEL
LIN {X 0,Y 367.909,Z 709.42,A -85,B 0,C 180,E1 15345.101,E2 15345.101} C_VEL
LIN {X 0,Y 362.315,Z 690.981,A -85,B 0,C 180,E1 15342.54,E2 15342.54} C_VEL
LIN {X 0,Y 358.876,Z 670.524,A -85,B 0,C 180,E1 15339.851,E2 15339.851} C_VEL
LIN {X 0,Y 357.895,Z 649.283,A -85,B 0,C 180,E1 15337.232,E2 15337.232} C_VEL
LIN {X 0,Y 359.408,Z 625.954,A -85,B 0,C 180,E1 15334.569,E2 15334.569} C_VEL
LIN {X 0,Y 363.781,Z 598.717,A -85,B 0,C 180,E1 15331.717,E2 15331.717} C_VEL
LIN {X 0,Y 366.667,Z 583.628,A -85,B 0,C 180,E1 15330.185,E2 15330.185} C_VEL
LIN {X 0,Y 358.614,Z 565.572,A -85,B 0,C 180,E1 15326.493,E2 15326.493} C_VEL
LIN {X 0,Y 350.001,Z 547.149,A -85,B 0,C 180,E1 15322.33,E2 15322.33} C_VEL
LIN {X 0,Y 342.341,Z 531.337,A -85,B 0,C 180,E1 15318.386,E2 15318.386} C_VEL
LIN {X 0,Y 335.241,Z 517.218,A -85,B 0,C 180,E1 15314.509,E2 15314.509} C_VEL
LIN {X 0,Y 328.756,Z 504.507,A -85,B 0,C 180,E1 15310.691,E2 15310.691} C_VEL
LIN {X 0,Y 323.533,Z 494.669,A -85,B 0,C 180,E1 15307.458,E2 15307.458} C_VEL
LIN {X 0,Y 321.127,Z 490.115,A -85,B 0,C 180,E1 15305.897,E2 15305.897} C_VEL
LIN {X 0,Y 318.801,Z 485.654,A -85,B 0,C 180,E1 15304.317,E2 15304.317} C_VEL
LIN {X 0,Y 316.986,Z 482.338,A -85,B 0,C 180,E1 15303.074,E2 15303.074} C_VEL
LIN {X 0,Y 316.249,Z 480.85,A -85,B 0,C 180,E1 15302.537,E2 15302.537} C_VEL
LIN {X 0,Y 314.428,Z 477.604,A -85,B 0,C 180,E1 15301.275,E2 15301.275} C_VEL
LIN {X 0,Y 314.167,Z 476.347,A -85,B 0,C 180,E1 15300.82,E2 15300.82} C_VEL
LIN {X 0,Y 314.159,Z 476.349,A -85,B 0,C 180,E1 15296.533,E2 15296.533} C_VEL
LIN {X 0,Y 314.158,Z 476.321,A -85,B 0,C 180,E1 15291.806,E2 15291.806} C_VEL
LIN {X 0,Y 314.132,Z 476.328,A -85,B 0,C 180,E1 15287.5,E2 15287.5} C_VEL
LIN {X 0,Y 314.173,Z 476.329,A -85,B 0,C 180,E1 15282.975,E2 15282.975} C_VEL
LIN {X 0,Y 314.174,Z 476.432,A -85,B 0,C 180,E1 15279.855,E2 15279.855} C_VEL
LIN {X 0,Y 315.144,Z 479.344,A -85,B 0,C 180,E1 15278.796,E2 15278.796} C_VEL
LIN {X 0,Y 317.859,Z 482.142,A -85,B 0,C 180,E1 15277.042,E2 15277.042} C_VEL
LIN {X 0,Y 318.331,Z 482.967,A -85,B 0,C 180,E1 15276.686,E2 15276.686} C_VEL
LIN {X 0,Y 320.234,Z 486.552,A -85,B 0,C 180,E1 15275.267,E2 15275.267} C_VEL
LIN {X 0,Y 321.785,Z 487.978,A -85,B 0,C 180,E1 15274.411,E2 15274.411} C_VEL
LIN {X 0,Y 323.78,Z 491.955,A -85,B 0,C 180,E1 15273.002,E2 15273.002} C_VEL
LIN {X 0,Y 325.322,Z 493.967,A -85,B 0,C 180,E1 15272.149,E2 15272.149} C_VEL
LIN {X 0,Y 327.961,Z 498.257,A -85,B 0,C 180,E1 15270.604,E2 15270.604} C_VEL
LIN {X 0,Y 331.93,Z 505.226,A -85,B 0,C 180,E1 15268.39,E2 15268.39} C_VEL
LIN {X 0,Y 334.198,Z 508.582,A -85,B 0,C 180,E1 15267.416,E2 15267.416} C_VEL
LIN {X 0,Y 343.829,Z 521.899,A -85,B 0,C 180,E1 15264.488,E2 15264.488} C_VEL
LIN {X 0,Y 353.23,Z 536.034,A -85,B 0,C 180,E1 15261.923,E2 15261.923} C_VEL
LIN {X 0,Y 362.469,Z 551.3,A -85,B 0,C 180,E1 15259.617,E2 15259.617} C_VEL
LIN {X 0,Y 368.886,Z 563.116,A -85,B 0,C 180,E1 15258.107,E2 15258.107} C_VEL
LIN {X 0,Y 358.968,Z 766.969,A -85,B 0,C 180,E1 15253.963,E2 15253.963} C_VEL
LIN {X 0,Y 357.134,Z 787.363,A -85,B 0,C 180,E1 15253.301,E2 15253.301} C_VEL
LIN {X 0,Y 354.448,Z 808.01,A -85,B 0,C 180,E1 15252.347,E2 15252.347} C_VEL
LIN {X 0,Y 351.355,Z 826.667,A -85,B 0,C 180,E1 15251.206,E2 15251.206} C_VEL
LIN {X 0,Y 347.662,Z 845.116,A -85,B 0,C 180,E1 15249.783,E2 15249.783} C_VEL
LIN {X 0,Y 343.326,Z 863.619,A -85,B 0,C 180,E1 15247.999,E2 15247.999} C_VEL
LIN {X 0,Y 338.801,Z 880.719,A -85,B 0,C 180,E1 15245.963,E2 15245.963} C_VEL
LIN {X 0,Y 334.289,Z 896.365,A -85,B 0,C 180,E1 15243.698,E2 15243.698} C_VEL
LIN {X 0,Y 329.924,Z 910.625,A -85,B 0,C 180,E1 15241.212,E2 15241.212} C_VEL
LIN {X 0,Y 325.732,Z 923.961,A -85,B 0,C 180,E1 15238.409,E2 15238.409} C_VEL
LIN {X 0,Y 321.898,Z 936.064,A -85,B 0,C 180,E1 15235.326,E2 15235.326} C_VEL
LIN {X 0,Y 318.73,Z 946.408,A -85,B 0,C 180,E1 15232.112,E2 15232.112} C_VEL
LIN {X 0,Y 316.017,Z 955.862,A -85,B 0,C 180,E1 15228.444,E2 15228.444} C_VEL
LIN {X 0,Y 314.149,Z 963.281,A -85,B 0,C 180,E1 15224.75,E2 15224.75} C_VEL
LIN {X 0,Y 313,Z 968.875,A -85,B 0,C 180,E1 15221.049,E2 15221.049} C_VEL
LIN {X 0,Y 312.404,Z 972.791,A -85,B 0,C 180,E1 15217.354,E2 15217.354} C_VEL
LIN {X 0,Y 312.16,Z 975.137,A -85,B 0,C 180,E1 15213.672,E2 15213.672} C_VEL
LIN {X 0,Y 312.115,Z 975.936,A -85,B 0,C 180,E1 15210.183,E2 15210.183} C_VEL
LIN {X 0,Y 312.144,Z 975.304,A -85,B 0,C 180,E1 15206.694,E2 15206.694} C_VEL
LIN {X 0,Y 312.365,Z 973.183,A -85,B 0,C 180,E1 15203.013,E2 15203.013} C_VEL
LIN {X 0,Y 312.899,Z 969.496,A -85,B 0,C 180,E1 15199.318,E2 15199.318} C_VEL
LIN {X 0,Y 313.971,Z 964.114,A -85,B 0,C 180,E1 15195.616,E2 15195.616} C_VEL
LIN {X 0,Y 315.746,Z 956.887,A -85,B 0,C 180,E1 15191.92,E2 15191.92} C_VEL
LIN {X 0,Y 318.197,Z 948.182,A -85,B 0,C 180,E1 15188.428,E2 15188.428} C_VEL
LIN {X 0,Y 320.266,Z 941.408,A -85,B 0,C 180,E1 15186.148,E2 15186.148} C_VEL
LIN {X 0,Y 320.548,Z 937.732,A -85,B 0,C 180,E1 15184.926,E2 15184.926} C_VEL
LIN {X 0,Y 318.289,Z 928.1,A -85,B 0,C 180,E1 15181.785,E2 15181.785} C_VEL
LIN {X 0,Y 318.875,Z 923.711,A -85,B 0,C 180,E1 15180.631,E2 15180.631} C_VEL
LIN {X 0,Y 323.211,Z 910.598,A -85,B 0,C 180,E1 15177.852,E2 15177.852} C_VEL
LIN {X 0,Y 327.965,Z 895.703,A -85,B 0,C 180,E1 15175.241,E2 15175.241} C_VEL
LIN {X 0,Y 332.777,Z 879.631,A -85,B 0,C 180,E1 15172.923,E2 15172.923} C_VEL
LIN {X 0,Y 337.325,Z 863.019,A -85,B 0,C 180,E1 15170.95,E2 15170.95} C_VEL
LIN {X 0,Y 341.588,Z 845.517,A -85,B 0,C 180,E1 15169.25,E2 15169.25} C_VEL
LIN {X 0,Y 345.432,Z 827.056,A -85,B 0,C 180,E1 15167.814,E2 15167.814} C_VEL
LIN {X 0,Y 348.737,Z 807.8,A -85,B 0,C 180,E1 15166.632,E2 15166.632} C_VEL
LIN {X 0,Y 351.475,Z 787.314,A -85,B 0,C 180,E1 15165.687,E2 15165.687} C_VEL
LIN {X 0,Y 353.373,Z 766.624,A -85,B 0,C 180,E1 15165.018,E2 15165.018} C_VEL
LIN {X 0,Y 363.139,Z 571.498,A -85,B 0,C 180,E1 15160.994,E2 15160.994} C_VEL
LIN {X 0,Y 356.973,Z 560.138,A -85,B 0,C 180,E1 15159.481,E2 15159.481} C_VEL
LIN {X 0,Y 353.736,Z 561.11,A -85,B 0,C 180,E1 15158.866,E2 15158.866} C_VEL
LIN {X 0,Y 349.6,Z 562.285,A -85,B 0,C 180,E1 15158.049,E2 15158.049} C_VEL
LIN {X 0,Y 345.686,Z 564.999,A -85,B 0,C 180,E1 15157.298,E2 15157.298} C_VEL
LIN {X 0,Y 344.571,Z 565.642,A -85,B 0,C 180,E1 15157.074,E2 15157.074} C_VEL
LIN {X 0,Y 339.755,Z 572.32,A -85,B 0,C 180,E1 15156.213,E2 15156.213} C_VEL
LIN {X 0,Y 336.065,Z 575.736,A -85,B 0,C 180,E1 15155.462,E2 15155.462} C_VEL
LIN {X 0,Y 334.29,Z 576.257,A -85,B 0,C 180,E1 15155.049,E2 15155.049} C_VEL
LIN {X 0,Y 333.835,Z 576.196,A -85,B 0,C 180,E1 15154.92,E2 15154.92} C_VEL
LIN {X 0,Y 328.873,Z 612.101,A -85,B 0,C 180,E1 15150.311,E2 15150.311} C_VEL
LIN {X 0,Y 325.99,Z 636.245,A -85,B 0,C 180,E1 15147.304,E2 15147.304} C_VEL
LIN {X 0,Y 326.159,Z 642.146,A -85,B 0,C 180,E1 15147.05,E2 15147.05} C_VEL
LIN {X 0,Y 318.097,Z 759.013,A -85,B 0,C 180,E1 15142.794,E2 15142.794} C_VEL
LIN {X 0,Y 316.981,Z 785.773,A -85,B 0,C 180,E1 15141.633,E2 15141.633} C_VEL
LIN {X 0,Y 316.053,Z 801.444,A -85,B 0,C 180,E1 15140.655,E2 15140.655} C_VEL
LIN {X 0,Y 314.695,Z 818.706,A -85,B 0,C 180,E1 15139.199,E2 15139.199} C_VEL
LIN {X 0,Y 313.25,Z 833.699,A -85,B 0,C 180,E1 15137.556,E2 15137.556} C_VEL
LIN {X 0,Y 311.742,Z 847.814,A -85,B 0,C 180,E1 15135.63,E2 15135.63} C_VEL
LIN {X 0,Y 310.26,Z 860.814,A -85,B 0,C 180,E1 15133.417,E2 15133.417} C_VEL
LIN {X 0,Y 308.965,Z 872.244,A -85,B 0,C 180,E1 15131.008,E2 15131.008} C_VEL
LIN {X 0,Y 307.861,Z 882.866,A -85,B 0,C 180,E1 15128.216,E2 15128.216} C_VEL
LIN {X 0,Y 307.096,Z 891.707,A -85,B 0,C 180,E1 15125.231,E2 15125.231} C_VEL
LIN {X 0,Y 306.744,Z 898.061,A -85,B 0,C 180,E1 15122.429,E2 15122.429} C_VEL
LIN {X 0,Y 306.721,Z 903.28,A -85,B 0,C 180,E1 15119.253,E2 15119.253} C_VEL
LIN {X 0,Y 307.085,Z 906.512,A -85,B 0,C 180,E1 15116.08,E2 15116.08} C_VEL
LIN {X 0,Y 307.825,Z 907.893,A -85,B 0,C 180,E1 15113.098,E2 15113.098} C_VEL
LIN {X 0,Y 309.177,Z 907.51,A -85,B 0,C 180,E1 15109.755,E2 15109.755} C_VEL
LIN {X 0,Y 311.18,Z 905.044,A -85,B 0,C 180,E1 15106.435,E2 15106.435} C_VEL
LIN {X 0,Y 313.731,Z 900.778,A -85,B 0,C 180,E1 15103.332,E2 15103.332} C_VEL
LIN {X 0,Y 316.769,Z 894.902,A -85,B 0,C 180,E1 15100.453,E2 15100.453} C_VEL
LIN {X 0,Y 320.214,Z 887.603,A -85,B 0,C 180,E1 15097.802,E2 15097.802} C_VEL
LIN {X 0,Y 324.243,Z 878.288,A -85,B 0,C 180,E1 15095.205,E2 15095.205} C_VEL
LIN {X 0,Y 328.527,Z 867.429,A -85,B 0,C 180,E1 15092.838,E2 15092.838} C_VEL
LIN {X 0,Y 333.32,Z 853.914,A -85,B 0,C 180,E1 15090.531,E2 15090.531} C_VEL
LIN {X 0,Y 337.93,Z 839.804,A -85,B 0,C 180,E1 15088.618,E2 15088.618} C_VEL
LIN {X 0,Y 342.627,Z 824.112,A -85,B 0,C 180,E1 15086.927,E2 15086.927} C_VEL
LIN {X 0,Y 349.351,Z 802.626,A -85,B 0,C 180,E1 15085.082,E2 15085.082} C_VEL
LIN {X 0,Y 359.014,Z 776.295,A -85,B 0,C 180,E1 15083.218,E2 15083.218} C_VEL
LIN {X 0,Y 369.112,Z 748.359,A -85,B 0,C 180,E1 15081.661,E2 15081.661} C_VEL
LIN {X 0,Y 378.452,Z 718.742,A -85,B 0,C 180,E1 15080.281,E2 15080.281} C_VEL
LIN {X 0,Y 379.923,Z 713.675,A -85,B 0,C 180,E1 15080.048,E2 15080.048} C_VEL
LIN {X 0,Y 378.545,Z 723.566,A -85,B 0,C 180,E1 15077.66,E2 15077.66} C_VEL
LIN {X 0,Y 378.445,Z 724.452,A -85,B 0,C 180,E1 15077.53,E2 15077.53} C_VEL
LIN {X 0,Y 375.249,Z 736.274,A -85,B 0,C 180,E1 15077.378,E2 15077.378} C_VEL
LIN {X 0,Y 369.032,Z 757.243,A -85,B 0,C 180,E1 15077.017,E2 15077.017} C_VEL
LIN {X 0,Y 363.327,Z 775.07,A -85,B 0,C 180,E1 15076.482,E2 15076.482} C_VEL
LIN {X 0,Y 357.042,Z 794.258,A -85,B 0,C 180,E1 15075.571,E2 15075.571} C_VEL
LIN {X 0,Y 349.164,Z 817.844,A -85,B 0,C 180,E1 15074.165,E2 15074.165} C_VEL
LIN {X 0,Y 345.993,Z 838.085,A -85,B 0,C 180,E1 15073.228,E2 15073.228} C_VEL
LIN {X 0,Y 342.39,Z 856.718,A -85,B 0,C 180,E1 15072.083,E2 15072.083} C_VEL
LIN {X 0,Y 338.12,Z 875.777,A -85,B 0,C 180,E1 15070.585,E2 15070.585} C_VEL
LIN {X 0,Y 333.467,Z 894.114,A -85,B 0,C 180,E1 15068.779,E2 15068.779} C_VEL
LIN {X 0,Y 328.669,Z 911.184,A -85,B 0,C 180,E1 15066.712,E2 15066.712} C_VEL
LIN {X 0,Y 323.839,Z 927.473,A -85,B 0,C 180,E1 15064.297,E2 15064.297} C_VEL
LIN {X 0,Y 319.105,Z 942.715,A -85,B 0,C 180,E1 15061.542,E2 15061.542} C_VEL
LIN {X 0,Y 315.004,Z 955.91,A -85,B 0,C 180,E1 15058.64,E2 15058.64} C_VEL
LIN {X 0,Y 311.411,Z 967.822,A -85,B 0,C 180,E1 15055.484,E2 15055.484} C_VEL
LIN {X 0,Y 308.383,Z 978.907,A -85,B 0,C 180,E1 15051.893,E2 15051.893} C_VEL
LIN {X 0,Y 306.178,Z 988.348,A -85,B 0,C 180,E1 15048.074,E2 15048.074} C_VEL
LIN {X 0,Y 304.858,Z 995.769,A -85,B 0,C 180,E1 15044.241,E2 15044.241} C_VEL
LIN {X 0,Y 304.285,Z 1001.129,A -85,B 0,C 180,E1 15040.605,E2 15040.605} C_VEL
LIN {X 0,Y 304.153,Z 1004.806,A -85,B 0,C 180,E1 15036.987,E2 15036.987} C_VEL
LIN {X 0,Y 304.24,Z 1006.975,A -85,B 0,C 180,E1 15033.392,E2 15033.392} C_VEL
LIN {X 0,Y 304.308,Z 1007.706,A -85,B 0,C 180,E1 15030.001,E2 15030.001} C_VEL
LIN {X 0,Y 304.236,Z 1006.971,A -85,B 0,C 180,E1 15026.61,E2 15026.61} C_VEL
LIN {X 0,Y 304.141,Z 1004.795,A -85,B 0,C 180,E1 15023.014,E2 15023.014} C_VEL
LIN {X 0,Y 304.273,Z 1001.118,A -85,B 0,C 180,E1 15019.397,E2 15019.397} C_VEL
LIN {X 0,Y 304.878,Z 995.442,A -85,B 0,C 180,E1 15015.568,E2 15015.568} C_VEL
LIN {X 0,Y 306.168,Z 988.192,A -85,B 0,C 180,E1 15011.864,E2 15011.864} C_VEL
LIN {X 0,Y 308.344,Z 978.873,A -85,B 0,C 180,E1 15008.106,E2 15008.106} C_VEL
LIN {X 0,Y 311.45,Z 967.504,A -85,B 0,C 180,E1 15004.435,E2 15004.435} C_VEL
LIN {X 0,Y 315.184,Z 955.072,A -85,B 0,C 180,E1 15001.173,E2 15001.173} C_VEL
LIN {X 0,Y 319.349,Z 941.659,A -85,B 0,C 180,E1 14998.266,E2 14998.266} C_VEL
LIN {X 0,Y 323.945,Z 926.853,A -85,B 0,C 180,E1 14995.611,E2 14995.611} C_VEL
LIN {X 0,Y 328.988,Z 909.852,A -85,B 0,C 180,E1 14993.114,E2 14993.114} C_VEL
LIN {X 0,Y 333.847,Z 892.33,A -85,B 0,C 180,E1 14991.029,E2 14991.029} C_VEL
LIN {X 0,Y 338.27,Z 874.71,A -85,B 0,C 180,E1 14989.327,E2 14989.327} C_VEL
LIN {X 0,Y 342.447,Z 855.916,A -85,B 0,C 180,E1 14987.869,E2 14987.869} C_VEL
LIN {X 0,Y 346.275,Z 835.68,A -85,B 0,C 180,E1 14986.654,E2 14986.654} C_VEL
LIN {X 0,Y 349.273,Z 815.866,A -85,B 0,C 180,E1 14985.766,E2 14985.766} C_VEL
LIN {X 0,Y 351.512,Z 794.942,A -85,B 0,C 180,E1 14985.106,E2 14985.106} C_VEL
LIN {X 0,Y 353.18,Z 769.814,A -85,B 0,C 180,E1 14984.607,E2 14984.607} C_VEL
LIN {X 0,Y 356.647,Z 739.373,A -85,B 0,C 180,E1 14984.317,E2 14984.317} C_VEL
LIN {X 0,Y 361.294,Z 711.78,A -85,B 0,C 180,E1 14984.301,E2 14984.301} C_VEL
LIN {X 0,Y 357.699,Z 703.232,A -85,B 0,C 180,E1 14983.443,E2 14983.443} C_VEL
LIN {X 0,Y 353.344,Z 684.093,A -85,B 0,C 180,E1 14980.818,E2 14980.818} C_VEL
LIN {X 0,Y 351.211,Z 663.551,A -85,B 0,C 180,E1 14978.153,E2 14978.153} C_VEL
LIN {X 0,Y 351.462,Z 641.435,A -85,B 0,C 180,E1 14975.475,E2 14975.475} C_VEL
LIN {X 0,Y 354.46,Z 615.641,A -85,B 0,C 180,E1 14972.6,E2 14972.6} C_VEL
LIN {X 0,Y 360.012,Z 587.279,A -85,B 0,C 180,E1 14969.673,E2 14969.673} C_VEL
LIN {X 0,Y 352.011,Z 569.287,A -85,B 0,C 180,E1 14965.939,E2 14965.939} C_VEL
LIN {X 0,Y 343.736,Z 551.498,A -85,B 0,C 180,E1 14961.859,E2 14961.859} C_VEL
LIN {X 0,Y 336.392,Z 536.283,A -85,B 0,C 180,E1 14958.006,E2 14958.006} C_VEL
LIN {X 0,Y 329.317,Z 522.133,A -85,B 0,C 180,E1 14954.057,E2 14954.057} C_VEL
LIN {X 0,Y 323.098,Z 509.888,A -85,B 0,C 180,E1 14950.34,E2 14950.34} C_VEL
LIN {X 0,Y 317.85,Z 499.971,A -85,B 0,C 180,E1 14947.047,E2 14947.047} C_VEL
LIN {X 0,Y 315.456,Z 495.435,A -85,B 0,C 180,E1 14945.456,E2 14945.456} C_VEL
LIN {X 0,Y 313.385,Z 491.394,A -85,B 0,C 180,E1 14944.025,E2 14944.025} C_VEL
LIN {X 0,Y 310.789,Z 486.566,A -85,B 0,C 180,E1 14942.212,E2 14942.212} C_VEL
LIN {X 0,Y 308.985,Z 483.002,A -85,B 0,C 180,E1 14940.855,E2 14940.855} C_VEL
LIN {X 0,Y 307.953,Z 481.392,A -85,B 0,C 180,E1 14940.17,E2 14940.17} C_VEL
LIN {X 0,Y 306.362,Z 478.059,A -85,B 0,C 180,E1 14938.878,E2 14938.878} C_VEL
LIN {X 0,Y 306.236,Z 477.335,A -85,B 0,C 180,E1 14938.597,E2 14938.597} C_VEL
LIN {X 0,Y 306.193,Z 477.333,A -85,B 0,C 180,E1 14934.002,E2 14934.002} C_VEL
LIN {X 0,Y 306.227,Z 477.341,A -85,B 0,C 180,E1 14929.654,E2 14929.654} C_VEL
LIN {X 0,Y 306.223,Z 477.334,A -85,B 0,C 180,E1 14924.858,E2 14924.858} C_VEL
LIN {X 0,Y 306.222,Z 477.344,A -85,B 0,C 180,E1 14924.081,E2 14924.081} C_VEL
LIN {X 0,Y 307.378,Z 480.545,A -85,B 0,C 180,E1 14922.586,E2 14922.586} C_VEL
LIN {X 0,Y 310.191,Z 483.277,A -85,B 0,C 180,E1 14920.413,E2 14920.413} C_VEL
LIN {X 0,Y 310.752,Z 484.493,A -85,B 0,C 180,E1 14919.862,E2 14919.862} C_VEL
LIN {X 0,Y 312.703,Z 487.877,A -85,B 0,C 180,E1 14918.228,E2 14918.228} C_VEL
LIN {X 0,Y 314.368,Z 489.392,A -85,B 0,C 180,E1 14917.168,E2 14917.168} C_VEL
LIN {X 0,Y 316.138,Z 493.065,A -85,B 0,C 180,E1 14915.722,E2 14915.722} C_VEL
LIN {X 0,Y 317.915,Z 495.004,A -85,B 0,C 180,E1 14914.676,E2 14914.676} C_VEL
LIN {X 0,Y 320.245,Z 499.203,A -85,B 0,C 180,E1 14913.082,E2 14913.082} C_VEL
LIN {X 0,Y 321.4,Z 500.982,A -85,B 0,C 180,E1 14912.384,E2 14912.384} C_VEL
LIN {X 0,Y 324.596,Z 506.375,A -85,B 0,C 180,E1 14910.472,E2 14910.472} C_VEL
LIN {X 0,Y 326.823,Z 509.557,A -85,B 0,C 180,E1 14909.479,E2 14909.479} C_VEL
LIN {X 0,Y 334.872,Z 520.341,A -85,B 0,C 180,E1 14906.777,E2 14906.777} C_VEL
LIN {X 0,Y 344.35,Z 534.153,A -85,B 0,C 180,E1 14903.934,E2 14903.934} C_VEL
LIN {X 0,Y 353.15,Z 548.013,A -85,B 0,C 180,E1 14901.551,E2 14901.551} C_VEL
LIN {X 0,Y 362.66,Z 564.837,A -85,B 0,C 180,E1 14899.174,E2 14899.174} C_VEL
LIN {X 0,Y 363.424,Z 566.668,A -85,B 0,C 180,E1 14898.979,E2 14898.979} C_VEL
LIN {X 0,Y 353.25,Z 767.395,A -85,B 0,C 180,E1 14894.861,E2 14894.861} C_VEL
LIN {X 0,Y 351.344,Z 787.84,A -85,B 0,C 180,E1 14894.191,E2 14894.191} C_VEL
LIN {X 0,Y 348.567,Z 808.44,A -85,B 0,C 180,E1 14893.231,E2 14893.231} C_VEL
LIN {X 0,Y 345.144,Z 828.16,A -85,B 0,C 180,E1 14892.004,E2 14892.004} C_VEL
LIN {X 0,Y 341.315,Z 846.393,A -85,B 0,C 180,E1 14890.566,E2 14890.566} C_VEL
LIN {X 0,Y 336.861,Z 864.641,A -85,B 0,C 180,E1 14888.775,E2 14888.775} C_VEL
LIN {X 0,Y 332.126,Z 881.778,A -85,B 0,C 180,E1 14886.696,E2 14886.696} C_VEL
LIN {X 0,Y 327.427,Z 897.317,A -85,B 0,C 180,E1 14884.396,E2 14884.396} C_VEL
LIN {X 0,Y 322.728,Z 911.941,A -85,B 0,C 180,E1 14881.781,E2 14881.781} C_VEL
LIN {X 0,Y 318.362,Z 925.126,A -85,B 0,C 180,E1 14878.923,E2 14878.923} C_VEL
LIN {X 0,Y 314.422,Z 936.926,A -85,B 0,C 180,E1 14875.826,E2 14875.826} C_VEL
LIN {X 0,Y 311.051,Z 947.337,A -85,B 0,C 180,E1 14872.489,E2 14872.489} C_VEL
LIN {X 0,Y 308.213,Z 956.705,A -85,B 0,C 180,E1 14868.732,E2 14868.732} C_VEL
LIN {X 0,Y 306.226,Z 964.16,A -85,B 0,C 180,E1 14864.878,E2 14864.878} C_VEL
LIN {X 0,Y 305.045,Z 969.535,A -85,B 0,C 180,E1 14861.149,E2 14861.149} C_VEL
LIN {X 0,Y 304.421,Z 973.358,A -85,B 0,C 180,E1 14857.358,E2 14857.358} C_VEL
LIN {X 0,Y 304.168,Z 975.614,A -85,B 0,C 180,E1 14853.58,E2 14853.58} C_VEL
LIN {X 0,Y 304.131,Z 976.368,A -85,B 0,C 180,E1 14849.999,E2 14849.999} C_VEL
LIN {X 0,Y 304.166,Z 975.651,A -85,B 0,C 180,E1 14846.418,E2 14846.418} C_VEL
LIN {X 0,Y 304.415,Z 973.443,A -85,B 0,C 180,E1 14842.639,E2 14842.639} C_VEL
LIN {X 0,Y 305.026,Z 969.665,A -85,B 0,C 180,E1 14838.848,E2 14838.848} C_VEL
LIN {X 0,Y 306.222,Z 964.216,A -85,B 0,C 180,E1 14835.051,E2 14835.051} C_VEL
LIN {X 0,Y 308.162,Z 956.911,A -85,B 0,C 180,E1 14831.263,E2 14831.263} C_VEL
LIN {X 0,Y 310.819,Z 948.098,A -85,B 0,C 180,E1 14827.691,E2 14827.691} C_VEL
LIN {X 0,Y 314.129,Z 937.864,A -85,B 0,C 180,E1 14824.348,E2 14824.348} C_VEL
LIN {X 0,Y 318.013,Z 926.262,A -85,B 0,C 180,E1 14821.245,E2 14821.245} C_VEL
LIN {X 0,Y 318.875,Z 923.711,A -85,B 0,C 180,E1 14820.631,E2 14820.631} C_VEL
LIN {X 0,Y 319.545,Z 919.23,A -85,B 0,C 180,E1 14819.499,E2 14819.499} C_VEL
LIN {X 0,Y 318.323,Z 907.763,A -85,B 0,C 180,E1 14816.543,E2 14816.543} C_VEL
LIN {X 0,Y 319.233,Z 902.583,A -85,B 0,C 180,E1 14815.507,E2 14815.507} C_VEL
LIN {X 0,Y 324.242,Z 887.019,A -85,B 0,C 180,E1 14813.034,E2 14813.034} C_VEL
LIN {X 0,Y 329.247,Z 870.069,A -85,B 0,C 180,E1 14810.826,E2 14810.826} C_VEL
LIN {X 0,Y 333.821,Z 852.934,A -85,B 0,C 180,E1 14809.007,E2 14809.007} C_VEL
LIN {X 0,Y 338.084,Z 834.577,A -85,B 0,C 180,E1 14807.426,E2 14807.426} C_VEL
LIN {X 0,Y 341.927,Z 814.605,A -85,B 0,C 180,E1 14806.07,E2 14806.07} C_VEL
LIN {X 0,Y 345.064,Z 793.78,A -85,B 0,C 180,E1 14805.006,E2 14805.006} C_VEL
LIN {X 0,Y 347.265,Z 773.334,A -85,B 0,C 180,E1 14804.264,E2 14804.264} C_VEL
LIN {X 0,Y 348.878,Z 747.624,A -85,B 0,C 180,E1 14803.657,E2 14803.657} C_VEL
LIN {X 0,Y 357.743,Z 574.741,A -85,B 0,C 180,E1 14800.082,E2 14800.082} C_VEL
LIN {X 0,Y 354.581,Z 568.689,A -85,B 0,C 180,E1 14799.276,E2 14799.276} C_VEL
LIN {X 0,Y 350.227,Z 570.14,A -85,B 0,C 180,E1 14798.437,E2 14798.437} C_VEL
LIN {X 0,Y 346.438,Z 572.82,A -85,B 0,C 180,E1 14797.724,E2 14797.724} C_VEL
LIN {X 0,Y 341.27,Z 579.448,A -85,B 0,C 180,E1 14796.809,E2 14796.809} C_VEL
LIN {X 0,Y 337.072,Z 583.095,A -85,B 0,C 180,E1 14795.968,E2 14795.968} C_VEL
LIN {X 0,Y 335.138,Z 584.275,A -85,B 0,C 180,E1 14795.549,E2 14795.549} C_VEL
LIN {X 0,Y 330.184,Z 591.61,A -85,B 0,C 180,E1 14794.596,E2 14794.596} C_VEL
LIN {X 0,Y 326.448,Z 595.385,A -85,B 0,C 180,E1 14793.774,E2 14793.774} C_VEL
LIN {X 0,Y 324.461,Z 596.018,A -85,B 0,C 180,E1 14793.266,E2 14793.266} C_VEL
LIN {X 0,Y 324.241,Z 596.129,A -85,B 0,C 180,E1 14793.186,E2 14793.186} C_VEL
LIN {X 0,Y 319.482,Z 631.55,A -85,B 0,C 180,E1 14788.61,E2 14788.61} C_VEL
LIN {X 0,Y 318.84,Z 637.326,A -85,B 0,C 180,E1 14787.916,E2 14787.916} C_VEL
LIN {X 0,Y 318.956,Z 643.08,A -85,B 0,C 180,E1 14787.662,E2 14787.662} C_VEL
LIN {X 0,Y 311.379,Z 745.499,A -85,B 0,C 180,E1 14783.835,E2 14783.835} C_VEL
LIN {X 0,Y 309.415,Z 785.25,A -85,B 0,C 180,E1 14782.128,E2 14782.128} C_VEL
LIN {X 0,Y 308.422,Z 801.8,A -85,B 0,C 180,E1 14781.091,E2 14781.091} C_VEL
LIN {X 0,Y 307.097,Z 818.232,A -85,B 0,C 180,E1 14779.693,E2 14779.693} C_VEL
LIN {X 0,Y 305.675,Z 832.808,A -85,B 0,C 180,E1 14778.104,E2 14778.104} C_VEL
LIN {X 0,Y 304.018,Z 847.831,A -85,B 0,C 180,E1 14776.037,E2 14776.037} C_VEL
LIN {X 0,Y 302.467,Z 861.028,A -85,B 0,C 180,E1 14773.769,E2 14773.769} C_VEL
LIN {X 0,Y 301.12,Z 872.703,A -85,B 0,C 180,E1 14771.298,E2 14771.298} C_VEL
LIN {X 0,Y 299.967,Z 883.502,A -85,B 0,C 180,E1 14768.434,E2 14768.434} C_VEL
LIN {X 0,Y 299.211,Z 892.021,A -85,B 0,C 180,E1 14765.561,E2 14765.561} C_VEL
LIN {X 0,Y 298.81,Z 899.038,A -85,B 0,C 180,E1 14762.493,E2 14762.493} C_VEL
LIN {X 0,Y 298.795,Z 904.394,A -85,B 0,C 180,E1 14759.233,E2 14759.233} C_VEL
LIN {X 0,Y 299.163,Z 907.67,A -85,B 0,C 180,E1 14756.168,E2 14756.168} C_VEL
LIN {X 0,Y 300.004,Z 909.383,A -85,B 0,C 180,E1 14752.917,E2 14752.917} C_VEL
LIN {X 0,Y 301.46,Z 909.163,A -85,B 0,C 180,E1 14749.49,E2 14749.49} C_VEL
LIN {X 0,Y 303.476,Z 907.108,A -85,B 0,C 180,E1 14746.278,E2 14746.278} C_VEL
LIN {X 0,Y 305.994,Z 903.5,A -85,B 0,C 180,E1 14743.289,E2 14743.289} C_VEL
LIN {X 0,Y 309.385,Z 897.772,A -85,B 0,C 180,E1 14740.164,E2 14740.164} C_VEL
LIN {X 0,Y 313.541,Z 889.865,A -85,B 0,C 180,E1 14737.105,E2 14737.105} C_VEL
LIN {X 0,Y 318.164,Z 880.14,A -85,B 0,C 180,E1 14734.299,E2 14734.299} C_VEL
LIN {X 0,Y 323.131,Z 868.638,A -85,B 0,C 180,E1 14731.743,E2 14731.743} C_VEL
LIN {X 0,Y 328.175,Z 855.956,A -85,B 0,C 180,E1 14729.518,E2 14729.518} C_VEL
LIN {X 0,Y 333.629,Z 841.161,A -85,B 0,C 180,E1 14727.456,E2 14727.456} C_VEL
LIN {X 0,Y 339.282,Z 824.561,A -85,B 0,C 180,E1 14725.643,E2 14725.643} C_VEL
LIN {X 0,Y 347.374,Z 802.772,A -85,B 0,C 180,E1 14723.737,E2 14723.737} C_VEL
LIN {X 0,Y 357.734,Z 777.482,A -85,B 0,C 180,E1 14721.954,E2 14721.954} C_VEL
LIN {X 0,Y 368.267,Z 750.407,A -85,B 0,C 180,E1 14720.466,E2 14720.466} C_VEL
LIN {X 0,Y 376.598,Z 725.753,A -85,B 0,C 180,E1 14719.323,E2 14719.323} C_VEL
LIN {X 0,Y 376.159,Z 728.621,A -85,B 0,C 180,E1 14718.649,E2 14718.649} C_VEL
LIN {X 0,Y 369.753,Z 749.762,A -85,B 0,C 180,E1 14718.392,E2 14718.392} C_VEL
LIN {X 0,Y 362.698,Z 770.751,A -85,B 0,C 180,E1 14717.866,E2 14717.866} C_VEL
LIN {X 0,Y 356.651,Z 787.859,A -85,B 0,C 180,E1 14717.149,E2 14717.149} C_VEL
LIN {X 0,Y 346.579,Z 814.981,A -85,B 0,C 180,E1 14715.564,E2 14715.564} C_VEL
LIN {X 0,Y 341.96,Z 827.256,A -85,B 0,C 180,E1 14714.685,E2 14714.685} C_VEL
LIN {X 0,Y 338.349,Z 847.12,A -85,B 0,C 180,E1 14713.615,E2 14713.615} C_VEL
LIN {X 0,Y 334.299,Z 865.852,A -85,B 0,C 180,E1 14712.297,E2 14712.297} C_VEL
LIN {X 0,Y 329.557,Z 884.876,A -85,B 0,C 180,E1 14710.602,E2 14710.602} C_VEL
LIN {X 0,Y 324.73,Z 902.189,A -85,B 0,C 180,E1 14708.687,E2 14708.687} C_VEL
LIN {X 0,Y 319.728,Z 918.694,A -85,B 0,C 180,E1 14706.455,E2 14706.455} C_VEL
LIN {X 0,Y 314.613,Z 934.741,A -85,B 0,C 180,E1 14703.792,E2 14703.792} C_VEL
LIN {X 0,Y 309.869,Z 949.146,A -85,B 0,C 180,E1 14700.868,E2 14700.868} C_VEL
LIN {X 0,Y 305.682,Z 962.06,A -85,B 0,C 180,E1 14697.677,E2 14697.677} C_VEL
LIN {X 0,Y 302.165,Z 973.513,A -85,B 0,C 180,E1 14694.226,E2 14694.226} C_VEL
LIN {X 0,Y 299.415,Z 983.473,A -85,B 0,C 180,E1 14690.527,E2 14690.527} C_VEL
LIN {X 0,Y 297.547,Z 991.878,A -85,B 0,C 180,E1 14686.598,E2 14686.598} C_VEL
LIN {X 0,Y 296.571,Z 998.097,A -85,B 0,C 180,E1 14682.858,E2 14682.858} C_VEL
LIN {X 0,Y 296.188,Z 1002.858,A -85,B 0,C 180,E1 14678.934,E2 14678.934} C_VEL
LIN {X 0,Y 296.19,Z 1005.72,A -85,B 0,C 180,E1 14675.231,E2 14675.231} C_VEL
LIN {X 0,Y 296.295,Z 1007.113,A -85,B 0,C 180,E1 14671.548,E2 14671.548} C_VEL
LIN {X 0,Y 296.29,Z 1007.088,A -85,B 0,C 180,E1 14668.261,E2 14668.261} C_VEL
LIN {X 0,Y 296.18,Z 1005.593,A -85,B 0,C 180,E1 14664.577,E2 14664.577} C_VEL
LIN {X 0,Y 296.178,Z 1002.63,A -85,B 0,C 180,E1 14660.872,E2 14660.872} C_VEL
LIN {X 0,Y 296.568,Z 997.882,A -85,B 0,C 180,E1 14656.992,E2 14656.992} C_VEL
LIN {X 0,Y 297.594,Z 991.495,A -85,B 0,C 180,E1 14653.206,E2 14653.206} C_VEL
LIN {X 0,Y 299.388,Z 983.442,A -85,B 0,C 180,E1 14649.473,E2 14649.473} C_VEL
LIN {X 0,Y 302.115,Z 973.47,A -85,B 0,C 180,E1 14645.772,E2 14645.772} C_VEL
LIN {X 0,Y 305.63,Z 962.006,A -85,B 0,C 180,E1 14642.32,E2 14642.32} C_VEL
LIN {X 0,Y 309.818,Z 949.079,A -85,B 0,C 180,E1 14639.128,E2 14639.128} C_VEL
LIN {X 0,Y 314.551,Z 934.656,A -85,B 0,C 180,E1 14636.203,E2 14636.203} C_VEL
LIN {X 0,Y 319.672,Z 918.596,A -85,B 0,C 180,E1 14633.54,E2 14633.54} C_VEL
LIN {X 0,Y 324.657,Z 902.068,A -85,B 0,C 180,E1 14631.305,E2 14631.305} C_VEL
LIN {X 0,Y 329.487,Z 884.722,A -85,B 0,C 180,E1 14629.39,E2 14629.39} C_VEL
LIN {X 0,Y 334.232,Z 865.651,A -85,B 0,C 180,E1 14627.695,E2 14627.695} C_VEL
LIN {X 0,Y 338.319,Z 846.665,A -85,B 0,C 180,E1 14626.365,E2 14626.365} C_VEL
LIN {X 0,Y 341.88,Z 826.853,A -85,B 0,C 180,E1 14625.304,E2 14625.304} C_VEL
LIN {X 0,Y 344.757,Z 806.1,A -85,B 0,C 180,E1 14624.5,E2 14624.5} C_VEL
LIN {X 0,Y 346.564,Z 784.258,A -85,B 0,C 180,E1 14623.92,E2 14623.92} C_VEL
LIN {X 0,Y 348.6,Z 759.449,A -85,B 0,C 180,E1 14623.545,E2 14623.545} C_VEL
LIN {X 0,Y 352.107,Z 732.441,A -85,B 0,C 180,E1 14623.362,E2 14623.362} C_VEL
LIN {X 0,Y 355.253,Z 713.994,A -85,B 0,C 180,E1 14623.366,E2 14623.366} C_VEL
LIN {X 0,Y 348.186,Z 696.179,A -85,B 0,C 180,E1 14621.596,E2 14621.596} C_VEL
LIN {X 0,Y 347.286,Z 692.406,A -85,B 0,C 180,E1 14621.137,E2 14621.137} C_VEL
LIN {X 0,Y 344.54,Z 671.054,A -85,B 0,C 180,E1 14618.285,E2 14618.285} C_VEL
LIN {X 0,Y 344.366,Z 648.827,A -85,B 0,C 180,E1 14615.499,E2 14615.499} C_VEL
LIN {X 0,Y 346.862,Z 623.858,A -85,B 0,C 180,E1 14612.618,E2 14612.618} C_VEL
LIN {X 0,Y 353.273,Z 590.748,A -85,B 0,C 180,E1 14609.131,E2 14609.131} C_VEL
LIN {X 0,Y 345.407,Z 572.94,A -85,B 0,C 180,E1 14605.367,E2 14605.367} C_VEL
LIN {X 0,Y 337.152,Z 555.205,A -85,B 0,C 180,E1 14601.211,E2 14601.211} C_VEL
LIN {X 0,Y 330.117,Z 540.619,A -85,B 0,C 180,E1 14597.448,E2 14597.448} C_VEL
LIN {X 0,Y 323.345,Z 526.956,A -85,B 0,C 180,E1 14593.592,E2 14593.592} C_VEL
LIN {X 0,Y 317.41,Z 515.214,A -85,B 0,C 180,E1 14589.977,E2 14589.977} C_VEL
LIN {X 0,Y 312.172,Z 505.225,A -85,B 0,C 180,E1 14586.621,E2 14586.621} C_VEL
LIN {X 0,Y 310.034,Z 501.133,A -85,B 0,C 180,E1 14585.181,E2 14585.181} C_VEL
LIN {X 0,Y 307.659,Z 496.662,A -85,B 0,C 180,E1 14583.54,E2 14583.54} C_VEL
LIN {X 0,Y 305.352,Z 492.25,A -85,B 0,C 180,E1 14581.876,E2 14581.876} C_VEL
LIN {X 0,Y 302.952,Z 487.624,A -85,B 0,C 180,E1 14580.082,E2 14580.082} C_VEL
LIN {X 0,Y 301.043,Z 483.922,A -85,B 0,C 180,E1 14578.595,E2 14578.595} C_VEL
LIN {X 0,Y 298.577,Z 479.689,A -85,B 0,C 180,E1 14576.736,E2 14576.736} C_VEL
LIN {X 0,Y 298.268,Z 478.327,A -85,B 0,C 180,E1 14576.252,E2 14576.252} C_VEL
LIN {X 0,Y 298.291,Z 478.298,A -85,B 0,C 180,E1 14571.42,E2 14571.42} C_VEL
LIN {X 0,Y 298.311,Z 478.453,A -85,B 0,C 180,E1 14570.157,E2 14570.157} C_VEL
LIN {X 0,Y 299.667,Z 481.938,A -85,B 0,C 180,E1 14567.67,E2 14567.67} C_VEL
LIN {X 0,Y 302.953,Z 484.843,A -85,B 0,C 180,E1 14564.298,E2 14564.298} C_VEL
LIN {X 0,Y 304.508,Z 488.358,A -85,B 0,C 180,E1 14562.417,E2 14562.417} C_VEL
LIN {X 0,Y 307.022,Z 490.947,A -85,B 0,C 180,E1 14560.401,E2 14560.401} C_VEL
LIN {X 0,Y 308.787,Z 494.478,A -85,B 0,C 180,E1 14558.736,E2 14558.736} C_VEL
LIN {X 0,Y 310.657,Z 496.426,A -85,B 0,C 180,E1 14557.473,E2 14557.473} C_VEL
LIN {X 0,Y 312.702,Z 500.315,A -85,B 0,C 180,E1 14555.84,E2 14555.84} C_VEL
LIN {X 0,Y 314.121,Z 502.029,A -85,B 0,C 180,E1 14554.954,E2 14554.954} C_VEL
LIN {X 0,Y 316.777,Z 506.455,A -85,B 0,C 180,E1 14553.169,E2 14553.169} C_VEL
LIN {X 0,Y 318.895,Z 509.978,A -85,B 0,C 180,E1 14551.996,E2 14551.996} C_VEL
LIN {X 0,Y 322.89,Z 515.007,A -85,B 0,C 180,E1 14550.453,E2 14550.453} C_VEL
LIN {X 0,Y 329.326,Z 523.615,A -85,B 0,C 180,E1 14548.162,E2 14548.162} C_VEL
LIN {X 0,Y 337.495,Z 535.281,A -85,B 0,C 180,E1 14545.538,E2 14545.538} C_VEL
LIN {X 0,Y 346.288,Z 548.972,A -85,B 0,C 180,E1 14542.985,E2 14542.985} C_VEL
LIN {X 0,Y 355.047,Z 564.062,A -85,B 0,C 180,E1 14540.655,E2 14540.655} C_VEL
LIN {X 0,Y 358.065,Z 569.919,A -85,B 0,C 180,E1 14539.885,E2 14539.885} C_VEL
LIN {X 0,Y 347.622,Z 767.824,A -85,B 0,C 180,E1 14535.788,E2 14535.788} C_VEL
LIN {X 0,Y 345.655,Z 788.206,A -85,B 0,C 180,E1 14535.115,E2 14535.115} C_VEL
LIN {X 0,Y 342.77,Z 808.874,A -85,B 0,C 180,E1 14534.145,E2 14534.145} C_VEL
LIN {X 0,Y 339.229,Z 828.552,A -85,B 0,C 180,E1 14532.91,E2 14532.91} C_VEL
LIN {X 0,Y 335.253,Z 846.792,A -85,B 0,C 180,E1 14531.459,E2 14531.459} C_VEL
LIN {X 0,Y 330.625,Z 865.045,A -85,B 0,C 180,E1 14529.649,E2 14529.649} C_VEL
LIN {X 0,Y 325.506,Z 882.836,A -85,B 0,C 180,E1 14527.458,E2 14527.458} C_VEL
LIN {X 0,Y 320.347,Z 899.135,A -85,B 0,C 180,E1 14524.984,E2 14524.984} C_VEL
LIN {X 0,Y 315.564,Z 913.258,A -85,B 0,C 180,E1 14522.375,E2 14522.375} C_VEL
LIN {X 0,Y 311.019,Z 926.292,A -85,B 0,C 180,E1 14519.462,E2 14519.462} C_VEL
LIN {X 0,Y 306.691,Z 938.577,A -85,B 0,C 180,E1 14516.11,E2 14516.11} C_VEL
LIN {X 0,Y 303.212,Z 948.752,A -85,B 0,C 180,E1 14512.693,E2 14512.693} C_VEL
LIN {X 0,Y 300.412,Z 957.515,A -85,B 0,C 180,E1 14509.036,E2 14509.036} C_VEL
LIN {X 0,Y 298.36,Z 964.788,A -85,B 0,C 180,E1 14505.152,E2 14505.152} C_VEL
LIN {X 0,Y 297.092,Z 970.195,A -85,B 0,C 180,E1 14501.255,E2 14501.255} C_VEL
LIN {X 0,Y 296.439,Z 973.925,A -85,B 0,C 180,E1 14497.363,E2 14497.363} C_VEL
LIN {X 0,Y 296.177,Z 976.091,A -85,B 0,C 180,E1 14493.483,E2 14493.483} C_VEL
LIN {X 0,Y 296.135,Z 976.771,A -85,B 0,C 180,E1 14489.806,E2 14489.806} C_VEL
LIN {X 0,Y 296.189,Z 975.998,A -85,B 0,C 180,E1 14486.128,E2 14486.128} C_VEL
LIN {X 0,Y 296.472,Z 973.703,A -85,B 0,C 180,E1 14482.246,E2 14482.246} C_VEL
LIN {X 0,Y 297.19,Z 969.704,A -85,B 0,C 180,E1 14478.248,E2 14478.248} C_VEL
LIN {X 0,Y 298.494,Z 964.289,A -85,B 0,C 180,E1 14474.455,E2 14474.455} C_VEL
LIN {X 0,Y 300.618,Z 956.924,A -85,B 0,C 180,E1 14470.572,E2 14470.572} C_VEL
LIN {X 0,Y 303.671,Z 947.514,A -85,B 0,C 180,E1 14466.726,E2 14466.726} C_VEL
LIN {X 0,Y 307.497,Z 936.424,A -85,B 0,C 180,E1 14463.129,E2 14463.129} C_VEL
LIN {X 0,Y 311.715,Z 924.423,A -85,B 0,C 180,E1 14459.973,E2 14459.973} C_VEL
LIN {X 0,Y 316.383,Z 911.005,A -85,B 0,C 180,E1 14457.072,E2 14457.072} C_VEL
LIN {X 0,Y 319.233,Z 902.583,A -85,B 0,C 180,E1 14455.507,E2 14455.507} C_VEL
LIN {X 0,Y 320.203,Z 897.336,A -85,B 0,C 180,E1 14454.497,E2 14454.497} C_VEL
LIN {X 0,Y 319.722,Z 884.061,A -85,B 0,C 180,E1 14451.79,E2 14451.79} C_VEL
LIN {X 0,Y 320.725,Z 878.233,A -85,B 0,C 180,E1 14450.892,E2 14450.892} C_VEL
LIN {X 0,Y 325.815,Z 860.696,A -85,B 0,C 180,E1 14448.832,E2 14448.832} C_VEL
LIN {X 0,Y 330.482,Z 842.415,A -85,B 0,C 180,E1 14447.098,E2 14447.098} C_VEL
LIN {X 0,Y 334.436,Z 824.366,A -85,B 0,C 180,E1 14445.725,E2 14445.725} C_VEL
LIN {X 0,Y 337.89,Z 804.935,A -85,B 0,C 180,E1 14444.567,E2 14444.567} C_VEL
LIN {X 0,Y 340.614,Z 784.607,A -85,B 0,C 180,E1 14443.67,E2 14443.67} C_VEL
LIN {X 0,Y 342.467,Z 764.055,A -85,B 0,C 180,E1 14443.045,E2 14443.045} C_VEL
LIN {X 0,Y 352.521,Z 578.169,A -85,B 0,C 180,E1 14439.164,E2 14439.164} C_VEL
LIN {X 0,Y 351.868,Z 577.37,A -85,B 0,C 180,E1 14439.007,E2 14439.007} C_VEL
LIN {X 0,Y 348.451,Z 579.75,A -85,B 0,C 180,E1 14438.38,E2 14438.38} C_VEL
LIN {X 0,Y 342.826,Z 586.536,A -85,B 0,C 180,E1 14437.4,E2 14437.4} C_VEL
